// TwinCAT 3 PLC project FrameworkUnitTest
// ProgramVersion: 3.1.4026.24
// libraries:
//   [RobustSolution], * (BATW)
//   Tc2_MC2, * (Beckhoff Automation GmbH)
//   Tc2_Standard, * (Beckhoff Automation GmbH)
//   Tc2_System, * (Beckhoff Automation GmbH)
//   Tc2_Utilities, * (Beckhoff Automation GmbH)
//   Tc3_JsonXml, * (Beckhoff Automation GmbH)
//   TcUnit, * (www.tcunit.org)
// project tree:
//   DUTs/ E_FakeAxisOperation.TcDUT, ST_FakeAxisCall.TcDUT, ST_FakeAxisScriptStep.TcDUT, ST_ReferencePortTestBranch.TcDUT, ST_TestModuleFixture.TcDUT, ST_TestServiceParam.TcDUT
//   GVLs/ GVL_TestConfig.TcGVL, GVL_TestSymbols.TcGVL
//   Fakes/ FB_FakeAxis_BaseUnit.TcPOU, FB_FakeBaseUnit.TcPOU, FB_FakeHookValueReader.TcPOU, FB_FakeModuleConfigurationAdapter.TcPOU, FB_FakeModuleReferenceBindings.TcPOU, FB_FakeVariableNodeReader.TcPOU, FB_ReferencePortFixture.TcPOU, FB_TestApplicationConfigRoot.TcPOU, FB_TestableCarryoverSubStateService.TcPOU, FB_TestableHookModule.TcPOU, FB_TestableModuleBase.TcPOU, FB_TestableServiceBase.TcPOU, FB_TestCompositeService.TcPOU, FB_TestPackMLBase.TcPOU, FB_TestPackMLModeSet.TcPOU
//   POUs/Test Suites/BaseUnit/ FB_Axis_BaseUnitTests.TcPOU, FB_BaseUnitTests.TcPOU, FB_FakeAxis_BaseUnitTests.TcPOU
//   POUs/Test Suites/Configuration/ FB_ApplicationConfigRootTests.TcPOU, FB_ConfigValueSnapshotReaderTests.TcPOU, FB_LinkVariableManagerTests.TcPOU, FB_ModuleConfigurationManagerTests.TcPOU, FB_ModuleReferenceBindingContextTests.TcPOU, FB_ModuleTypeRegistryTests.TcPOU, FB_ReferenceManagerTests.TcPOU
//   POUs/Test Suites/Infrastructure/ FB_UtcClockTests.TcPOU
//   POUs/Test Suites/Module/ FB_ModuleAlarmManagerTests.TcPOU, FB_ModuleBaseTests.TcPOU
//   POUs/Test Suites/PackML/ FB_PackMLBaseTests.TcPOU, FB_PackMLModeSetTests.TcPOU
//   POUs/Test Suites/Service/ FB_CompositeServiceBaseTests.TcPOU, FB_ServiceBaseTests.TcPOU, FB_ServiceCallerTests.TcPOU, FB_ServiceCoordinatorTests.TcPOU, FB_ServiceExecuteSubStateTests.TcPOU, FB_SetMaterialServiceTests.TcPOU
//   / PlcTask.TcTTO
//   POUs/ TEST_PROG.TcPOU
// (motion and I/O tree: see PLC project robustsolutionframework)
// real-time tasks:
//   TASK UnitTest Task: cycle T#10ms, priority 21, ADS port 351
//   TASK DemoProject Task: cycle T#10ms, priority 22, ADS port 352
// variable links:

CONFIGURATION FrameworkUnitTest
    RESOURCE PLC ON TwinCAT3
        TASK PlcTask(INTERVAL := T#10ms, PRIORITY := 21);
        PROGRAM TEST_PROG WITH PlcTask : TEST_PROG;
    END_RESOURCE
END_CONFIGURATION

// ---- DUTs/E_FakeAxisOperation.TcDUT
{attribute 'qualified_only'}
{attribute 'to_string'}
TYPE E_FakeAxisOperation :
(
None := 0,
Jog,
MoveAbs,
MoveVel,
Stop,
Reset,
Halt
) UINT;
END_TYPE

// ---- DUTs/ST_FakeAxisCall.TcDUT
TYPE ST_FakeAxisCall :
STRUCT
Sequence : UDINT;
Cycle : UDINT;
Operation : E_FakeAxisOperation;
OwnerId : T_ResourceOwnerId;
Accepted : BOOL;
Execute : BOOL;
JogForward : BOOL;
JogBackwards : BOOL;
Mode : E_JogMode;
Direction : MC_Direction;
Position : LREAL;
Velocity : LREAL;
Acceleration : LREAL;
Deceleration : LREAL;
END_STRUCT
END_TYPE

// ---- DUTs/ST_FakeAxisScriptStep.TcDUT
TYPE ST_FakeAxisScriptStep :
STRUCT
Operation : E_FakeAxisOperation;
AfterActiveCycles : UINT;
Done : BOOL;
InVelocity : BOOL;
Error : BOOL;
ErrorId : UDINT;
Started : BOOL;
ResultLatched : BOOL;
Consumed : BOOL;
ActiveCycles : UINT;
END_STRUCT
END_TYPE

// ---- DUTs/ST_ReferencePortTestBranch.TcDUT
TYPE ST_ReferencePortTestBranch :
STRUCT
Axis : I_Axis_BaseUnit;
Axes : ARRAY[1..2] OF I_Axis_BaseUnit;
PortWithAnIntentionallyLongNameForReferenceBindingTests : I_Axis_BaseUnit;
END_STRUCT
END_TYPE

// ---- DUTs/ST_TestModuleFixture.TcDUT
TYPE ST_TestModuleFixture :
STRUCT
InputBool : BOOL;
OutputBool : BOOL;
SignedValue : DINT;
UnsignedValue : UDINT;
RealValue : REAL;
LongRealValue : LREAL;
TextValue : STRING(80);
BaseUnitPort : I_BaseUnit;
Nested : ST_ReferencePortTestBranch;
END_STRUCT
END_TYPE

// ---- DUTs/ST_TestServiceParam.TcDUT
TYPE ST_TestServiceParam :
STRUCT
// 使用兩個欄位，確保 Tc3_JsonXml 能反查真實 DUT 型別名稱。
Value : DINT;
Sequence : UDINT;
END_STRUCT
END_TYPE

// ---- GVLs/GVL_TestConfig.TcGVL
{attribute 'qualified_only'}
VAR_GLOBAL CONSTANT
// 預設不註冊需要外部 NC 與測試檔案的案例，避免把缺少前置條件誤報為成功。
RunNcAxisRuntimeTests : BOOL := FALSE;
RunConfigurationFileRuntimeTests : BOOL := TRUE;
ConfigurationFixtureRoot : STRING(255) := 'C:\ProgramData\RobustSolution\Tests\';
END_VAR

// ---- GVLs/GVL_TestSymbols.TcGVL
{attribute 'qualified_only'}
VAR_GLOBAL
// 具名全域變數會產生 ADS symbol，供 symbol/reflection 相關 runtime 測試使用。
InfrastructureBool : BOOL;
InfrastructureOutputBool : BOOL;
InfrastructureDInt : DINT;
InfrastructureLReal : LREAL;
InfrastructureText : STRING(80);
ModuleOne : ST_TestModuleFixture;
ModuleTwo : ST_TestModuleFixture;
RegisteredBaseUnit : FB_BaseUnit;
SecondaryBaseUnit : FB_BaseUnit;
UnprovidedBaseUnit : FB_FakeBaseUnit;
END_VAR

// ---- POUs/TEST_PROG.TcPOU
PROGRAM TEST_PROG
VAR
	BaseUnitTests : FB_BaseUnitTests;
	AxisBaseUnitTests : FB_Axis_BaseUnitTests;
	FakeAxisContractTests : FB_FakeAxis_BaseUnitTests;
	UtcClockTests : FB_UtcClockTests;
	PackMLBaseTests : FB_PackMLBaseTests;
	PackMLModeSetTests : FB_PackMLModeSetTests;
	ServiceBaseTests : FB_ServiceBaseTests;
	ServiceExecuteSubStateTests : FB_ServiceExecuteSubStateTests;
	CompositeServiceBaseTests : FB_CompositeServiceBaseTests;
	SetMaterialServiceTests : FB_SetMaterialServiceTests;
	ServiceCallerTests : FB_ServiceCallerTests;
	ServiceCoordinatorTests : FB_ServiceCoordinatorTests;
	ModuleAlarmManagerTests : FB_ModuleAlarmManagerTests;
	ModuleBaseTests : FB_ModuleBaseTests;
	ConfigValueSnapshotReaderTests : FB_ConfigValueSnapshotReaderTests;
	LinkVariableManagerTests : FB_LinkVariableManagerTests;
	ReferenceManagerTests : FB_ReferenceManagerTests;
	ModuleReferenceBindingContextTests : FB_ModuleReferenceBindingContextTests;
	ModuleTypeRegistryTests : FB_ModuleTypeRegistryTests;
	ModuleConfigurationManagerTests : FB_ModuleConfigurationManagerTests;
	ApplicationConfigRootTests : FB_ApplicationConfigRootTests;
END_VAR

// 上述 FB_TestSuite instances 會向 TcUnit 註冊；runner 每個週期統一驅動測試。
TcUnit.RUN();

END_PROGRAM

// ---- POUs/Test Suites/BaseUnit/FB_BaseUnitTests.TcPOU
FUNCTION_BLOCK FB_BaseUnitTests EXTENDS TcUnit.FB_TestSuite
VAR
	_BaseUnit : FB_BaseUnit;
END_VAR

InitialStateAndZeroOwnerAreSafe();
OwnershipIsExclusiveAndReleaseIsOwnerOnly();
AdsMetadataDescribesTheInstance();

METHOD InitialStateAndZeroOwnerAreSafe
TEST('InitialStateAndZeroOwnerAreSafe');

// Arrange：新建立的 BaseUnit 尚未被任何 Service 占用。
// Act / Assert：OwnerId=0 代表未占用，永遠不能取得、擁有或釋放資源。
AssertFalse(
	Condition := _BaseUnit.ResourceIsAcquired,
	Message := 'A new BaseUnit must be unowned.'
);
AssertTrue(
	Condition := _BaseUnit.ResourceOwnerId = 0,
	Message := 'The unowned sentinel must be zero.'
);
AssertFalse(
	Condition := _BaseUnit.M_AcquireResource(OwnerId := 0),
	Message := 'Owner zero must not acquire a resource.'
);
AssertFalse(
	Condition := _BaseUnit.M_IsResourceOwner(OwnerId := 0),
	Message := 'Owner zero must never be reported as owner.'
);
AssertFalse(
	Condition := _BaseUnit.M_ReleaseResource(OwnerId := 0),
	Message := 'Owner zero must not release a resource.'
);

TEST_FINISHED();
END_METHOD

METHOD OwnershipIsExclusiveAndReleaseIsOwnerOnly
TEST('OwnershipIsExclusiveAndReleaseIsOwnerOnly');

// Arrange / Act：Owner 11 先取得資源；同 Owner 重入應維持冪等。
AssertTrue(
	Condition := _BaseUnit.M_AcquireResource(OwnerId := 11),
	Message := 'The first valid owner must acquire the resource.'
);
AssertTrue(
	Condition := _BaseUnit.M_AcquireResource(OwnerId := 11),
	Message := 'Re-acquiring by the owner must be idempotent.'
);

// Assert：競爭者不能取得或釋放；目前 Owner 可正常釋放。
AssertFalse(
	Condition := _BaseUnit.M_AcquireResource(OwnerId := 12),
	Message := 'A competing owner must be rejected.'
);
AssertFalse(
	Condition := _BaseUnit.M_ReleaseResource(OwnerId := 12),
	Message := 'A non-owner must not release the resource.'
);
AssertTrue(
	Condition := _BaseUnit.ResourceIsAcquired AND (_BaseUnit.ResourceOwnerId = 11),
	Message := 'Rejected operations must preserve ownership.'
);
AssertTrue(
	Condition := _BaseUnit.M_ReleaseResource(OwnerId := 11),
	Message := 'The current owner must release the resource.'
);
AssertFalse(
	Condition := _BaseUnit.ResourceIsAcquired,
	Message := 'Release must restore the unowned state.'
);

TEST_FINISHED();
END_METHOD

METHOD AdsMetadataDescribesTheInstance
VAR
	pData : PVOID;
	nData : UDINT;
END_VAR
TEST('AdsMetadataDescribesTheInstance');

// Act：取得 framework 對外提供的 ADS metadata。
AssertTrue(
	Condition := _BaseUnit.M_GetAdsSymbolMetadata(Address => pData, Size => nData),
	Message := 'BaseUnit metadata must be available.'
);

// Assert：位址必須指向目前 instance，大小必須涵蓋整個 FB。
AssertTrue(
	Condition := pData = ADR(_BaseUnit),
	Message := 'Metadata address must identify this BaseUnit instance.'
);
AssertTrue(
	Condition := nData = SIZEOF(_BaseUnit),
	Message := 'Metadata size must match the BaseUnit instance.'
);

TEST_FINISHED();
END_METHOD

END_FUNCTION_BLOCK

// ---- POUs/Test Suites/BaseUnit/FB_Axis_BaseUnitTests.TcPOU
FUNCTION_BLOCK FB_Axis_BaseUnitTests EXTENDS TcUnit.FB_TestSuite
VAR
	_Axis : FB_Axis_BaseUnit;
END_VAR

AllMotionCommandsRejectNonOwners();
InitialAxisFeedbackIsNeutral();
NcAxisLifecycleRequiresExplicitRuntimeOptIn();

METHOD AllMotionCommandsRejectNonOwners
VAR
	bDone : BOOL;
	bInVelocity : BOOL;
	bError : BOOL;
	nErrorId : UDINT;
END_VAR
TEST('AllMotionCommandsRejectNonOwners');

// Arrange：不先取得 ownership，避免任何 MC function block 被啟動。
// Act / Assert：六種命令都必須在 ownership gate 被拒絕，輸出保持中性。
AssertFalse(
	Condition := _Axis.M_Halt(
		OwnerId := 1,
		Execute := TRUE,
		Deceleration := 1,
		Done => bDone,
		Error => bError
	),
	Message := 'Halt must reject a non-owner.'
);
AssertFalse(
	Condition := bDone OR bError,
	Message := 'Rejected Halt outputs must be neutral.'
);
AssertFalse(
	Condition := _Axis.M_Jog(
		OwnerId := 1,
		JogForward := TRUE,
		JogBackwards := FALSE,
		Mode := E_JogMode.MC_JOGMODE_CONTINOUS,
		Position := 0,
		Velocity := 1,
		Acceleration := 1,
		Deceleration := 1,
		Done => bDone,
		Error => bError,
		ErrorId => nErrorId
	),
	Message := 'Jog must reject a non-owner.'
);
AssertFalse(
	Condition := bDone OR bError OR (nErrorId <> 0),
	Message := 'Rejected Jog outputs must be neutral.'
);
AssertFalse(
	Condition := _Axis.M_MoveAbs(
		OwnerId := 1,
		Execute := TRUE,
		Position := 1,
		Velocity := 1,
		Acceleration := 1,
		Deceleration := 1,
		Done => bDone,
		Error => bError,
		ErrorId => nErrorId
	),
	Message := 'MoveAbs must reject a non-owner.'
);
AssertFalse(
	Condition := _Axis.M_MoveVel(
		OwnerId := 1,
		Execute := TRUE,
		Direction := MC_Direction.MC_Positive_Direction,
		Velocity := 1,
		Acceleration := 1,
		Deceleration := 1,
		InVelocity => bInVelocity,
		Error => bError
	),
	Message := 'MoveVel must reject a non-owner.'
);
AssertFalse(
	Condition := _Axis.M_Reset(
		OwnerId := 1,
		Execute := TRUE,
		Done => bDone,
		Error => bError,
		ErrorId => nErrorId
	),
	Message := 'Reset must reject a non-owner.'
);
AssertFalse(
	Condition := _Axis.M_Stop(
		OwnerId := 1,
		Execute := TRUE,
		Deceleration := 1,
		Done => bDone,
		Error => bError,
		ErrorId => nErrorId
	),
	Message := 'Stop must reject a non-owner.'
);

TEST_FINISHED();
END_METHOD

METHOD InitialAxisFeedbackIsNeutral
TEST('InitialAxisFeedbackIsNeutral');

// Assert：未連結 NC 軸時，只驗證不需驅動硬體的公開 feedback 初值。
AssertTrue(
	Condition := (_Axis.AxisActualPosition = 0.0) AND (_Axis.AxisActualVelocity = 0.0),
	Message := 'Unlinked Axis feedback must start at zero.'
);
AssertFalse(
	Condition := _Axis.AxisHasJob,
	Message := 'An unlinked Axis must not report a job.'
);

TEST_FINISHED();
END_METHOD

METHOD NcAxisLifecycleRequiresExplicitRuntimeOptIn
VAR
	bDone : BOOL;
	bError : BOOL;
	nErrorId : UDINT;
END_VAR
// RuntimeDependent：未在 XAE 將此 instance 的 _Axis 連到模擬 NC 軸時，不註冊這個 TcUnit case。
IF NOT GVL_TestConfig.RunNcAxisRuntimeTests THEN
	RETURN;
END_IF
TEST('NcAxisLifecycleRequiresExplicitRuntimeOptIn');

// Arrange：XAE 中已完成模擬 NC 軸連結，且測試開關明確設為 TRUE。
AssertTrue(
	Condition := _Axis.M_AcquireResource(OwnerId := 77),
	Message := 'Runtime owner must acquire the Axis.'
);

// Act：Reset 命令由真實 MC_Reset 執行；多掃描完成狀態由目標 Runtime 驗證。
AssertTrue(
	Condition := _Axis.M_Reset(
		OwnerId := 77,
		Execute := TRUE,
		Done => bDone,
		Error => bError,
		ErrorId => nErrorId
	),
	Message := 'Owned Reset must reach the MC layer.'
);
_Axis.M_CyclicUpdate();
AssertFalse(
	Condition := bDone AND bError,
	Message := 'MC Reset must never report Done and Error together.'
);

TEST_FINISHED();
END_METHOD

END_FUNCTION_BLOCK

// ---- POUs/Test Suites/BaseUnit/FB_FakeAxis_BaseUnitTests.TcPOU
FUNCTION_BLOCK FB_FakeAxis_BaseUnitTests EXTENDS TcUnit.FB_TestSuite
VAR
	_FakeAxis : FB_FakeAxis_BaseUnit;
	_Axis : I_Axis_BaseUnit;
END_VAR

ResourceCanBeAcquiredAndReleased();
OwnerZeroAndNonOwnerStopAreRejected();
AllNonOwnerMotionCommandsAreRejected();
ValidOwnerHaltIsAcceptedAndRecorded();
OwnerZeroAndNonOwnerHaltAreRejected();
HaltDoneIsPublishedAfterConfiguredCycles();
HaltErrorIsPublishedAfterConfiguredCycles();
HaltWithdrawalClearsResultAndPreservesOwnership();
ScriptAndHistoryOverflowAreExplicit();
CommandHistoryPreservesParameters();
ResponseRemainsLatchedUntilCommandWithdrawal();
JogErrorIsPublishedAfterConfiguredCycles();
ActualFeedbackIsAvailableThroughInterface();

METHOD ActualFeedbackIsAvailableThroughInterface
VAR
	FakeAxis : FB_FakeAxis_BaseUnit;
	Axis : I_Axis_BaseUnit;
END_VAR
TEST('ActualFeedbackIsAvailableThroughInterface');

FakeAxis.M_ResetScenario();
FakeAxis.M_SetAxisFeedback(ActualPosition := 45.25, ActualVelocity := 123.5);
Axis := FakeAxis;

AssertTrue(
	Condition := Axis.AxisActualPosition = 45.25,
	Message := 'Axis interface must expose actual position feedback.'
);
AssertTrue(
	Condition := Axis.AxisActualVelocity = 123.5,
	Message := 'Axis interface must expose actual velocity feedback.'
);

TEST_FINISHED();
END_METHOD

METHOD AllNonOwnerMotionCommandsAreRejected
VAR
	bDone : BOOL;
	bInVelocity : BOOL;
	bError : BOOL;
	nErrorId : UDINT;
END_VAR
TEST('AllNonOwnerMotionCommandsAreRejected');

_FakeAxis.M_ResetScenario();
_Axis := _FakeAxis;
AssertTrue(
	Condition := _Axis.M_AcquireResource(OwnerId := 1),
	Message := 'Owner 1 must acquire the Axis.'
);
AssertFalse(
	Condition := _Axis.M_Jog(
		OwnerId := 2,
		JogForward := TRUE,
		JogBackwards := FALSE,
		Mode := E_JogMode.MC_JOGMODE_CONTINOUS,
		Position := 1,
		Velocity := 2,
		Acceleration := 3,
		Deceleration := 4,
		Done => bDone,
		Error => bError,
		ErrorId => nErrorId
	),
	Message := 'Non-Owner Jog must be rejected.'
);
AssertFalse(
	Condition := bDone OR bError OR (nErrorId <> 0),
	Message := 'Rejected Jog outputs must be neutral.'
);
AssertFalse(
	Condition := _Axis.M_MoveAbs(
		OwnerId := 2,
		Execute := TRUE,
		Position := 1,
		Velocity := 2,
		Acceleration := 3,
		Deceleration := 4,
		Done => bDone,
		Error => bError
	),
	Message := 'Non-Owner MoveAbs must be rejected.'
);
AssertFalse(
	Condition := _Axis.M_MoveVel(
		OwnerId := 2,
		Execute := TRUE,
		Direction := MC_Direction.MC_Positive_Direction,
		Velocity := 2,
		Acceleration := 3,
		Deceleration := 4,
		InVelocity => bInVelocity,
		Error => bError
	),
	Message := 'Non-Owner MoveVel must be rejected.'
);
AssertFalse(
	Condition := _Axis.M_Reset(
		OwnerId := 2,
		Execute := TRUE,
		Done => bDone,
		Error => bError
	),
	Message := 'Non-Owner Reset must be rejected.'
);
AssertFalse(
	Condition := bDone OR bInVelocity OR bError,
	Message := 'All rejected motion outputs must remain neutral.'
);

TEST_FINISHED();
END_METHOD

METHOD CommandHistoryPreservesParameters
VAR
	CallRecord : ST_FakeAxisCall;
END_VAR
TEST('CommandHistoryPreservesParameters');

_FakeAxis.M_ResetScenario();
_Axis := _FakeAxis;
AssertTrue(
	Condition := _Axis.M_AcquireResource(OwnerId := 5),
	Message := 'History test Owner must acquire Axis.'
);
_Axis.M_MoveAbs(
	OwnerId := 5,
	Execute := TRUE,
	Position := 123.5,
	Velocity := 45.5,
	Acceleration := 67.5,
	Deceleration := 89.5
);
AssertTrue(
	Condition := _FakeAxis.M_GetCall(Index := 1, CallRecord => CallRecord),
	Message := 'Accepted MoveAbs must be present in history.'
);
AssertTrue(
	Condition := CallRecord.Accepted AND CallRecord.Execute,
	Message := 'History must retain acceptance and Execute.'
);
AssertTrue(
	Condition :=
		(CallRecord.Position = 123.5)
		AND (CallRecord.Velocity = 45.5)
		AND (CallRecord.Acceleration = 67.5)
		AND (CallRecord.Deceleration = 89.5),
	Message := 'History must retain all motion parameters.'
);

_Axis.M_MoveAbs(
	OwnerId := 6,
	Execute := FALSE,
	Position := 1,
	Velocity := 2,
	Acceleration := 3,
	Deceleration := 4
);
AssertTrue(
	Condition := _FakeAxis.M_GetCall(Index := 2, CallRecord => CallRecord),
	Message := 'Rejected command must still be recorded.'
);
AssertFalse(
	Condition := CallRecord.Accepted,
	Message := 'Rejected history entry must be marked rejected.'
);
AssertTrue(
	Condition := CallRecord.Sequence = 2,
	Message := 'History sequence must be global and monotonic.'
);

TEST_FINISHED();
END_METHOD

METHOD HaltDoneIsPublishedAfterConfiguredCycles
VAR_INST
	FakeAxis : FB_FakeAxis_BaseUnit;
	Axis : I_Axis_BaseUnit;
	nPhase : UINT;
	bDone : BOOL;
	bError : BOOL;
END_VAR
TEST('HaltDoneIsPublishedAfterConfiguredCycles');

CASE nPhase OF
	0:
		FakeAxis.M_ResetScenario();
		Axis := FakeAxis;
		AssertTrue(
			Condition := Axis.M_AcquireResource(OwnerId := 21),
			Message := 'Halt Done test Owner must acquire the Axis.'
		);
		AssertTrue(
			Condition := FakeAxis.M_QueueResult(
				Operation := E_FakeAxisOperation.Halt,
				AfterActiveCycles := 2,
				Done := TRUE,
				InVelocity := FALSE,
				Error := FALSE,
				ErrorId := 0
			),
			Message := 'Halt Done script must be queued.'
		);
		AssertTrue(
			Condition := Axis.M_Halt(
				OwnerId := 21,
				Execute := TRUE,
				Deceleration := 10,
				Done => bDone,
				Error => bError
			),
			Message := 'Owner Halt must be accepted.'
		);
		AssertFalse(
			Condition := bDone OR bError,
			Message := 'Halt result must initially be pending.'
		);
		nPhase := 1;

	1:
		Axis.M_CyclicUpdate();
		Axis.M_Halt(
			OwnerId := 21,
			Execute := TRUE,
			Deceleration := 10,
			Done => bDone,
			Error => bError
		);
		AssertFalse(
			Condition := bDone OR bError,
			Message := 'Halt Done must remain pending after one active cycle.'
		);
		nPhase := 2;

	2:
		Axis.M_CyclicUpdate();
		Axis.M_Halt(
			OwnerId := 21,
			Execute := TRUE,
			Deceleration := 10,
			Done => bDone,
			Error => bError
		);
		AssertTrue(
			Condition := bDone AND NOT bError,
			Message := 'Halt Done must be published on the configured cycle.'
		);
		nPhase := 0;
		TEST_FINISHED();
END_CASE
END_METHOD

METHOD HaltErrorIsPublishedAfterConfiguredCycles
VAR_INST
	FakeAxis : FB_FakeAxis_BaseUnit;
	Axis : I_Axis_BaseUnit;
	nPhase : UINT;
	bDone : BOOL;
	bError : BOOL;
END_VAR
TEST('HaltErrorIsPublishedAfterConfiguredCycles');

CASE nPhase OF
	0:
		FakeAxis.M_ResetScenario();
		Axis := FakeAxis;
		AssertTrue(
			Condition := Axis.M_AcquireResource(OwnerId := 22),
			Message := 'Halt Error test Owner must acquire the Axis.'
		);
		AssertTrue(
			Condition := FakeAxis.M_QueueResult(
				Operation := E_FakeAxisOperation.Halt,
				AfterActiveCycles := 2,
				Done := FALSE,
				InVelocity := FALSE,
				Error := TRUE,
				ErrorId := 16#5678
			),
			Message := 'Halt Error script must be queued.'
		);
		Axis.M_Halt(
			OwnerId := 22,
			Execute := TRUE,
			Deceleration := 11,
			Done => bDone,
			Error => bError
		);
		AssertFalse(
			Condition := bDone OR bError,
			Message := 'Halt Error must initially be pending.'
		);
		nPhase := 1;

	1:
		Axis.M_CyclicUpdate();
		Axis.M_Halt(
			OwnerId := 22,
			Execute := TRUE,
			Deceleration := 11,
			Done => bDone,
			Error => bError
		);
		AssertFalse(
			Condition := bDone OR bError,
			Message := 'Halt Error must remain pending after one active cycle.'
		);
		nPhase := 2;

	2:
		Axis.M_CyclicUpdate();
		Axis.M_Halt(
			OwnerId := 22,
			Execute := TRUE,
			Deceleration := 11,
			Done => bDone,
			Error => bError
		);
		AssertTrue(
			Condition := bError AND NOT bDone,
			Message := 'Halt Error must be published on the configured cycle.'
		);
		nPhase := 0;
		TEST_FINISHED();
END_CASE
END_METHOD

METHOD HaltWithdrawalClearsResultAndPreservesOwnership
VAR_INST
	FakeAxis : FB_FakeAxis_BaseUnit;
	Axis : I_Axis_BaseUnit;
	nPhase : UINT;
	bDone : BOOL;
	bError : BOOL;
	CallRecord : ST_FakeAxisCall;
END_VAR
TEST('HaltWithdrawalClearsResultAndPreservesOwnership');

CASE nPhase OF
	0:
		FakeAxis.M_ResetScenario();
		Axis := FakeAxis;
		AssertTrue(
			Condition := Axis.M_AcquireResource(OwnerId := 23),
			Message := 'Halt withdrawal test Owner must acquire the Axis.'
		);
		AssertTrue(
			Condition := FakeAxis.M_QueueResult(
				Operation := E_FakeAxisOperation.Halt,
				AfterActiveCycles := 1,
				Done := TRUE,
				InVelocity := FALSE,
				Error := FALSE,
				ErrorId := 0
			),
			Message := 'Halt withdrawal script must be queued.'
		);
		Axis.M_Halt(OwnerId := 23, Execute := TRUE, Deceleration := 12);
		nPhase := 1;

	1:
		Axis.M_CyclicUpdate();
		Axis.M_Halt(
			OwnerId := 23,
			Execute := TRUE,
			Deceleration := 12,
			Done => bDone,
			Error => bError
		);
		AssertTrue(
			Condition := bDone AND NOT bError,
			Message := 'Halt must complete before command withdrawal.'
		);
		AssertTrue(
			Condition := Axis.M_IsResourceOwner(OwnerId := 23),
			Message := 'Halt completion must not release its Owner.'
		);
		AssertTrue(
			Condition := Axis.M_Halt(OwnerId := 23, Execute := FALSE, Deceleration := 12),
			Message := 'Owner must be allowed to withdraw Halt.'
		);
		AssertTrue(
			Condition := FakeAxis.M_GetCall(Index := 3, CallRecord => CallRecord),
			Message := 'Withdrawn Halt must be recorded.'
		);
		AssertTrue(
			Condition :=
				(CallRecord.Operation = E_FakeAxisOperation.Halt)
				AND CallRecord.Accepted
				AND NOT CallRecord.Execute,
			Message := 'Halt history must expose accepted command withdrawal.'
		);
		Axis.M_CyclicUpdate();
		nPhase := 2;

	2:
		Axis.M_Halt(
			OwnerId := 23,
			Execute := FALSE,
			Deceleration := 12,
			Done => bDone,
			Error => bError
		);
		AssertFalse(
			Condition := bDone OR bError,
			Message := 'Halt result must clear after withdrawal and cyclic update.'
		);
		AssertTrue(
			Condition := Axis.M_IsResourceOwner(OwnerId := 23),
			Message := 'Halt withdrawal must preserve resource ownership.'
		);
		AssertFalse(
			Condition := Axis.M_AcquireResource(OwnerId := 24),
			Message := 'A contender must remain rejected after Halt withdrawal.'
		);
		nPhase := 0;
		TEST_FINISHED();
END_CASE
END_METHOD

METHOD JogErrorIsPublishedAfterConfiguredCycles
VAR_INST
	FakeAxis : FB_FakeAxis_BaseUnit;
	Axis : I_Axis_BaseUnit;
	nPhase : UINT;
	bError : BOOL;
	bQueued : BOOL;
END_VAR
TEST('JogErrorIsPublishedAfterConfiguredCycles');

CASE nPhase OF
	0:
		FakeAxis.M_ResetScenario();
		Axis := FakeAxis;
		AssertTrue(
			Condition := Axis.M_AcquireResource(OwnerId := 1),
			Message := 'Test Owner must acquire the Axis.'
		);
		bQueued := FakeAxis.M_QueueResult(
			Operation := E_FakeAxisOperation.Jog,
			AfterActiveCycles := 2,
			Done := FALSE,
			InVelocity := FALSE,
			Error := TRUE,
			ErrorId := 16#1234);
		AssertTrue(Condition := bQueued, Message := 'A valid Jog Error script must be queued.');
		Axis.M_Jog(
			OwnerId := 1,
			JogForward := TRUE,
			JogBackwards := FALSE,
			Mode := E_JogMode.MC_JOGMODE_CONTINOUS,
			Position := 0,
			Velocity := 10,
			Acceleration := 20,
			Deceleration := 30);
		nPhase := 1;

	1:
		Axis.M_CyclicUpdate();
		Axis.M_Jog(
			OwnerId := 1,
			JogForward := TRUE,
			JogBackwards := FALSE,
			Mode := E_JogMode.MC_JOGMODE_CONTINOUS,
			Position := 0,
			Velocity := 10,
			Acceleration := 20,
			Deceleration := 30,
			Error => bError);
		AssertFalse(
			Condition := bError,
			Message := 'Jog Error must remain pending after one active cycle.'
		);
		nPhase := 2;

	2:
		Axis.M_CyclicUpdate();
		Axis.M_Jog(
			OwnerId := 1,
			JogForward := TRUE,
			JogBackwards := FALSE,
			Mode := E_JogMode.MC_JOGMODE_CONTINOUS,
			Position := 0,
			Velocity := 10,
			Acceleration := 20,
			Deceleration := 30,
			Error => bError);
		AssertTrue(
			Condition := bError,
			Message := 'Jog Error must be published on the configured cycle.'
		);
		nPhase := 0;
		TEST_FINISHED();
END_CASE
END_METHOD

METHOD OwnerZeroAndNonOwnerHaltAreRejected
VAR
	bDone : BOOL;
	bError : BOOL;
	bAccepted : BOOL;
	CallRecord : ST_FakeAxisCall;
END_VAR
TEST('OwnerZeroAndNonOwnerHaltAreRejected');

_FakeAxis.M_ResetScenario();
_Axis := _FakeAxis;
AssertTrue(
	Condition := _Axis.M_AcquireResource(OwnerId := 31),
	Message := 'Valid Owner must acquire the Axis.'
);

bAccepted := _Axis.M_Halt(
	OwnerId := 0,
	Execute := TRUE,
	Deceleration := 20,
	Done => bDone,
	Error => bError
);
AssertFalse(Condition := bAccepted, Message := 'OwnerId zero Halt must be rejected.');
AssertFalse(
	Condition := bDone OR bError,
	Message := 'OwnerId zero Halt outputs must be neutral.'
);
AssertTrue(
	Condition := _FakeAxis.M_GetCall(Index := 1, CallRecord => CallRecord),
	Message := 'OwnerId zero Halt must be recorded.'
);
AssertFalse(
	Condition := CallRecord.Accepted,
	Message := 'OwnerId zero Halt history must be rejected.'
);

bAccepted := _Axis.M_Halt(
	OwnerId := 32,
	Execute := TRUE,
	Deceleration := 21,
	Done => bDone,
	Error => bError
);
AssertFalse(Condition := bAccepted, Message := 'Non-Owner Halt must be rejected.');
AssertFalse(
	Condition := bDone OR bError,
	Message := 'Non-Owner Halt outputs must be neutral.'
);
AssertTrue(
	Condition := _FakeAxis.M_GetCall(Index := 2, CallRecord => CallRecord),
	Message := 'Non-Owner Halt must be recorded.'
);
AssertFalse(
	Condition := CallRecord.Accepted,
	Message := 'Non-Owner Halt history must be rejected.'
);
AssertTrue(
	Condition := _Axis.M_IsResourceOwner(OwnerId := 31),
	Message := 'Rejected Halt must preserve the current Owner.'
);

TEST_FINISHED();
END_METHOD

METHOD OwnerZeroAndNonOwnerStopAreRejected
VAR
	bDone : BOOL;
	bError : BOOL;
	bRejected : BOOL;
	bAccepted : BOOL;
END_VAR
TEST('OwnerZeroAndNonOwnerStopAreRejected');

_FakeAxis.M_ResetScenario();
_Axis := _FakeAxis;
AssertFalse(
	Condition := _Axis.M_AcquireResource(OwnerId := 0),
	Message := 'OwnerId zero must never acquire a resource.'
);
AssertTrue(
	Condition := _Axis.M_AcquireResource(OwnerId := 1),
	Message := 'Valid Owner must acquire the Axis.'
);
AssertTrue(
	Condition := _FakeAxis.M_QueueResult(
		Operation := E_FakeAxisOperation.Stop,
		AfterActiveCycles := 1,
		Done := TRUE,
		InVelocity := FALSE,
		Error := FALSE,
		ErrorId := 0
	),
	Message := 'Stop Done script must be accepted.'
);

bAccepted := _Axis.M_Stop(OwnerId := 1, Execute := TRUE, Deceleration := 10);
bRejected := _Axis.M_Stop(
	OwnerId := 2,
	Execute := FALSE,
	Deceleration := 99,
	Done => bDone,
	Error => bError
);
AssertFalse(Condition := bRejected, Message := 'Non-Owner Stop must be rejected.');
AssertFalse(
	Condition := bDone OR bError,
	Message := 'Rejected Stop must return neutral outputs.'
);

_Axis.M_CyclicUpdate();
_Axis.M_Stop(
	OwnerId := 1,
	Execute := TRUE,
	Deceleration := 10,
	Done => bDone,
	Error => bError
);
AssertTrue(
	Condition := bAccepted AND bDone AND NOT bError,
	Message := 'Rejected Stop must not cancel the active Owner command.'
);

TEST_FINISHED();
END_METHOD

METHOD ResourceCanBeAcquiredAndReleased
VAR
	bAcquired : BOOL;
	bContenderAcquired : BOOL;
	bReleased : BOOL;
END_VAR
TEST('ResourceCanBeAcquiredAndReleased');

_FakeAxis.M_ResetScenario();
_Axis := _FakeAxis;

bAcquired := _Axis.M_AcquireResource(OwnerId := 1);
bContenderAcquired := _Axis.M_AcquireResource(OwnerId := 2);
bReleased := _Axis.M_ReleaseResource(OwnerId := 1);

AssertTrue(
	Condition := bAcquired,
	Message := 'The first valid Owner must acquire the Axis.'
);
AssertFalse(
	Condition := bContenderAcquired,
	Message := 'A competing Owner must be rejected.'
);
AssertTrue(Condition := bReleased, Message := 'The active Owner must release the Axis.');
AssertFalse(
	Condition := _Axis.M_IsResourceOwner(OwnerId := 1),
	Message := 'The Axis must be unowned after Release.'
);

TEST_FINISHED();
END_METHOD

METHOD ResponseRemainsLatchedUntilCommandWithdrawal
VAR
	bError : BOOL;
END_VAR
TEST('ResponseRemainsLatchedUntilCommandWithdrawal');

_FakeAxis.M_ResetScenario();
_Axis := _FakeAxis;
AssertTrue(
	Condition := _Axis.M_AcquireResource(OwnerId := 1),
	Message := 'Latch test Owner must acquire Axis.'
);
AssertTrue(
	Condition := _FakeAxis.M_QueueResult(
		Operation := E_FakeAxisOperation.Jog,
		AfterActiveCycles := 1,
		Done := FALSE,
		InVelocity := FALSE,
		Error := TRUE,
		ErrorId := 1
	),
	Message := 'Jog Error script must be queued.'
);
_Axis.M_Jog(
	OwnerId := 1,
	JogForward := TRUE,
	JogBackwards := FALSE,
	Mode := E_JogMode.MC_JOGMODE_CONTINOUS,
	Position := 0,
	Velocity := 1,
	Acceleration := 1,
	Deceleration := 1
);
_Axis.M_CyclicUpdate();
_Axis.M_Jog(
	OwnerId := 1,
	JogForward := TRUE,
	JogBackwards := FALSE,
	Mode := E_JogMode.MC_JOGMODE_CONTINOUS,
	Position := 0,
	Velocity := 1,
	Acceleration := 1,
	Deceleration := 1,
	Error => bError
);
AssertTrue(Condition := bError, Message := 'Configured Error must latch.');
_Axis.M_CyclicUpdate();
_Axis.M_Jog(
	OwnerId := 1,
	JogForward := TRUE,
	JogBackwards := FALSE,
	Mode := E_JogMode.MC_JOGMODE_CONTINOUS,
	Position := 0,
	Velocity := 1,
	Acceleration := 1,
	Deceleration := 1,
	Error => bError
);
AssertTrue(
	Condition := bError,
	Message := 'Error must remain latched while Jog remains active.'
);
_Axis.M_Jog(
	OwnerId := 1,
	JogForward := FALSE,
	JogBackwards := FALSE,
	Mode := E_JogMode.MC_JOGMODE_CONTINOUS,
	Position := 0,
	Velocity := 1,
	Acceleration := 1,
	Deceleration := 1
);
_Axis.M_CyclicUpdate();
_Axis.M_Jog(
	OwnerId := 1,
	JogForward := FALSE,
	JogBackwards := FALSE,
	Mode := E_JogMode.MC_JOGMODE_CONTINOUS,
	Position := 0,
	Velocity := 1,
	Acceleration := 1,
	Deceleration := 1,
	Error => bError
);
AssertFalse(
	Condition := bError,
	Message :=
		'Error must clear after both Jog directions are withdrawn and cyclic update runs.'
);

TEST_FINISHED();
END_METHOD

METHOD ScriptAndHistoryOverflowAreExplicit
VAR
	nIndex : UINT;
	bQueued : BOOL;
END_VAR
TEST('ScriptAndHistoryOverflowAreExplicit');

_FakeAxis.M_ResetScenario();
_Axis := _FakeAxis;
FOR nIndex := 1 TO 32 DO
	bQueued := _FakeAxis.M_QueueResult(
		Operation := E_FakeAxisOperation.MoveAbs,
		AfterActiveCycles := nIndex,
		Done := TRUE,
		InVelocity := FALSE,
		Error := FALSE,
		ErrorId := 0
	);
END_FOR
bQueued := _FakeAxis.M_QueueResult(
	Operation := E_FakeAxisOperation.MoveAbs,
	AfterActiveCycles := 33,
	Done := TRUE,
	InVelocity := FALSE,
	Error := FALSE,
	ErrorId := 0
);
AssertFalse(Condition := bQueued, Message := 'Script queue must reject entry 33.');
AssertTrue(
	Condition := _FakeAxis.ScriptOverflowed,
	Message := 'Script overflow must be visible.'
);

_FakeAxis.M_ResetScenario();
bQueued := _FakeAxis.M_QueueResult(
	Operation := E_FakeAxisOperation.Jog,
	AfterActiveCycles := 1,
	Done := TRUE,
	InVelocity := FALSE,
	Error := TRUE,
	ErrorId := 0
);
AssertFalse(
	Condition := bQueued,
	Message := 'Done and Error cannot be configured together.'
);
AssertTrue(
	Condition := _FakeAxis.ScriptConfigurationError,
	Message := 'Invalid script configuration must be visible.'
);

FOR nIndex := 1 TO 257 DO
	_Axis.M_Reset(OwnerId := 77, Execute := TRUE);
END_FOR
AssertTrue(
	Condition := _FakeAxis.HistoryCount = 256,
	Message := 'History must stop at its fixed capacity.'
);
AssertTrue(
	Condition := _FakeAxis.HistoryOverflowed,
	Message := 'History overflow must be visible and must not overwrite calls.'
);

TEST_FINISHED();
END_METHOD

METHOD ValidOwnerHaltIsAcceptedAndRecorded
VAR
	bDone : BOOL;
	bError : BOOL;
	CallRecord : ST_FakeAxisCall;
END_VAR
TEST('ValidOwnerHaltIsAcceptedAndRecorded');

_FakeAxis.M_ResetScenario();
_Axis := _FakeAxis;
AssertTrue(
	Condition := _Axis.M_AcquireResource(OwnerId := 11),
	Message := 'Valid Halt Owner must acquire the Axis.'
);
AssertTrue(
	Condition := _Axis.M_Halt(
		OwnerId := 11,
		Execute := TRUE,
		Deceleration := 12.5,
		Done => bDone,
		Error => bError
	),
	Message := 'Valid Owner Halt must be accepted.'
);
AssertFalse(
	Condition := bDone OR bError,
	Message := 'Unscripted Halt outputs must be neutral.'
);
AssertTrue(
	Condition := _FakeAxis.M_GetCall(Index := 1, CallRecord => CallRecord),
	Message := 'Accepted Halt must be present in history.'
);
AssertTrue(
	Condition :=
		(CallRecord.Operation = E_FakeAxisOperation.Halt)
		AND CallRecord.Accepted
		AND CallRecord.Execute,
	Message := 'History must identify an accepted active Halt.'
);
AssertTrue(
	Condition := (CallRecord.OwnerId = 11) AND (CallRecord.Deceleration = 12.5),
	Message := 'Halt history must preserve Owner and deceleration.'
);

TEST_FINISHED();
END_METHOD

END_FUNCTION_BLOCK

// ---- Fakes/FB_FakeAxis_BaseUnit.TcPOU
FUNCTION_BLOCK FB_FakeAxis_BaseUnit EXTENDS FB_BaseUnit IMPLEMENTS I_Axis_BaseUnit
VAR
	_bAxisIsDisabled : BOOL;
	_bAxisHasJob : BOOL;
	_fAxisActualPosition : LREAL;
	_fAxisActualVelocity : LREAL;
	_nCycle : UDINT;
	_nCallSequence : UDINT;

	_aScripts : ARRAY[1..32] OF ST_FakeAxisScriptStep;
	_nScriptCount : UINT;
	_bScriptOverflowed : BOOL;
	_bScriptConfigurationError : BOOL;

	_aHistory : ARRAY[1..256] OF ST_FakeAxisCall;
	_nHistoryCount : UINT;
	_bHistoryOverflowed : BOOL;

	_bJogActive : BOOL;
	_bMoveAbsActive : BOOL;
	_bMoveVelActive : BOOL;
	_bStopActive : BOOL;
	_bResetActive : BOOL;
	_bHaltActive : BOOL;

	_bJogDone : BOOL;
	_bJogInVelocity : BOOL;
	_bJogError : BOOL;
	_nJogErrorId : UDINT;
	_bMoveAbsDone : BOOL;
	_bMoveAbsInVelocity : BOOL;
	_bMoveAbsError : BOOL;
	_nMoveAbsErrorId : UDINT;
	_bMoveVelDone : BOOL;
	_bMoveVelInVelocity : BOOL;
	_bMoveVelError : BOOL;
	_nMoveVelErrorId : UDINT;
	_bStopDone : BOOL;
	_bStopInVelocity : BOOL;
	_bStopError : BOOL;
	_nStopErrorId : UDINT;
	_bResetDone : BOOL;
	_bResetInVelocity : BOOL;
	_bResetError : BOOL;
	_nResetErrorId : UDINT;
	_bHaltDone : BOOL;
	_bHaltInVelocity : BOOL;
	_bHaltError : BOOL;
	_nHaltErrorId : UDINT;
END_VAR

M_CyclicUpdate();

PROPERTY AxisActualPosition : LREAL
GET
AxisActualPosition := _fAxisActualPosition;
END_GET
END_PROPERTY

PROPERTY AxisActualVelocity : LREAL
GET
AxisActualVelocity := _fAxisActualVelocity;
END_GET
END_PROPERTY

PROPERTY AxisHasJob : BOOL
GET
AxisHasJob := _bAxisHasJob;
END_GET
END_PROPERTY

PROPERTY AxisIsDisabled : BOOL
GET
AxisIsDisabled := _bAxisIsDisabled;
END_GET
END_PROPERTY

PROPERTY CurrentCycle : UDINT
GET
CurrentCycle := _nCycle;
END_GET
END_PROPERTY

PROPERTY HistoryCount : UINT
GET
HistoryCount := _nHistoryCount;
END_GET
END_PROPERTY

PROPERTY HistoryOverflowed : BOOL
GET
HistoryOverflowed := _bHistoryOverflowed;
END_GET
END_PROPERTY

METHOD M_ClearCallHistory
VAR_INPUT
END_VAR
MEMSET(ADR(_aHistory), 0, SIZEOF(_aHistory));
_nHistoryCount := 0;
_nCallSequence := 0;
_bHistoryOverflowed := FALSE;
END_METHOD

METHOD M_CyclicUpdate
VAR_INPUT
END_VAR
_nCycle := _nCycle + 1;

M_ProcessOperation(
	Operation := E_FakeAxisOperation.Jog,
	Active := _bJogActive,
	Done := _bJogDone,
	InVelocity := _bJogInVelocity,
	Error := _bJogError,
	ErrorId := _nJogErrorId
);
M_ProcessOperation(
	Operation := E_FakeAxisOperation.MoveAbs,
	Active := _bMoveAbsActive,
	Done := _bMoveAbsDone,
	InVelocity := _bMoveAbsInVelocity,
	Error := _bMoveAbsError,
	ErrorId := _nMoveAbsErrorId
);
M_ProcessOperation(
	Operation := E_FakeAxisOperation.MoveVel,
	Active := _bMoveVelActive,
	Done := _bMoveVelDone,
	InVelocity := _bMoveVelInVelocity,
	Error := _bMoveVelError,
	ErrorId := _nMoveVelErrorId
);
M_ProcessOperation(
	Operation := E_FakeAxisOperation.Stop,
	Active := _bStopActive,
	Done := _bStopDone,
	InVelocity := _bStopInVelocity,
	Error := _bStopError,
	ErrorId := _nStopErrorId
);
M_ProcessOperation(
	Operation := E_FakeAxisOperation.Reset,
	Active := _bResetActive,
	Done := _bResetDone,
	InVelocity := _bResetInVelocity,
	Error := _bResetError,
	ErrorId := _nResetErrorId
);
M_ProcessOperation(
	Operation := E_FakeAxisOperation.Halt,
	Active := _bHaltActive,
	Done := _bHaltDone,
	InVelocity := _bHaltInVelocity,
	Error := _bHaltError,
	ErrorId := _nHaltErrorId
);
END_METHOD

METHOD M_GetCall : BOOL
VAR_INPUT
	Index : UINT;
END_VAR
VAR_OUTPUT
	CallRecord : ST_FakeAxisCall;
END_VAR
M_GetCall := FALSE;
MEMSET(ADR(CallRecord), 0, SIZEOF(CallRecord));
IF (Index = 0) OR (Index > _nHistoryCount) THEN
	RETURN;
END_IF
CallRecord := _aHistory[Index];
M_GetCall := TRUE;
END_METHOD

METHOD M_Halt : BOOL
VAR_INPUT
	OwnerId : T_ResourceOwnerId;
	Execute : BOOL;
	Deceleration : LREAL;
END_VAR
VAR_OUTPUT
	Done : BOOL;
	Error : BOOL;
END_VAR
VAR
	bAccepted : BOOL;
END_VAR
bAccepted := M_IsResourceOwner(OwnerId := OwnerId);
M_RecordCall(
	Operation := E_FakeAxisOperation.Halt,
	OwnerId := OwnerId,
	Accepted := bAccepted,
	Execute := Execute,
	JogForward := FALSE,
	JogBackwards := FALSE,
	Mode := E_JogMode.MC_JOGMODE_CONTINOUS,
	Direction := MC_Direction.MC_Positive_Direction,
	Position := 0,
	Velocity := 0,
	Acceleration := 0,
	Deceleration := Deceleration
);

M_Halt := bAccepted;
IF NOT bAccepted THEN
	Done := FALSE;
	Error := FALSE;
	RETURN;
END_IF

_bHaltActive := Execute;
Done := _bHaltDone;
Error := _bHaltError;
END_METHOD

METHOD M_Jog : BOOL
VAR_INPUT
	OwnerId : T_ResourceOwnerId;
	JogForward : BOOL;
	JogBackwards : BOOL;
	Mode : E_JogMode;
	Position : LREAL;
	Velocity : LREAL;
	Acceleration : LREAL;
	Deceleration : LREAL;
END_VAR
VAR_OUTPUT
	Done : BOOL;
	Error : BOOL;
	ErrorId : UDINT;
END_VAR
VAR
	bAccepted : BOOL;
END_VAR
bAccepted := M_IsResourceOwner(OwnerId := OwnerId);
M_RecordCall(
	Operation := E_FakeAxisOperation.Jog,
	OwnerId := OwnerId,
	Accepted := bAccepted,
	Execute := JogForward OR JogBackwards,
	JogForward := JogForward,
	JogBackwards := JogBackwards,
	Mode := Mode,
	Direction := MC_Direction.MC_Positive_Direction,
	Position := Position,
	Velocity := Velocity,
	Acceleration := Acceleration,
	Deceleration := Deceleration
);

M_Jog := bAccepted;
IF NOT bAccepted THEN
	Done := FALSE;
	Error := FALSE;
	ErrorId := 0;
	RETURN;
END_IF

_bJogActive := JogForward OR JogBackwards;
Done := _bJogDone;
Error := _bJogError;
ErrorId := _nJogErrorId;
END_METHOD

METHOD M_MoveAbs : BOOL
VAR_INPUT
	OwnerId : T_ResourceOwnerId;
	Execute : BOOL;
	Position : LREAL;
	Velocity : LREAL;
	Acceleration : LREAL;
	Deceleration : LREAL;
END_VAR
VAR_OUTPUT
	Done : BOOL;
	Error : BOOL;
	ErrorId : UDINT;
END_VAR
VAR
	bAccepted : BOOL;
END_VAR
bAccepted := M_IsResourceOwner(OwnerId := OwnerId);
M_RecordCall(
	Operation := E_FakeAxisOperation.MoveAbs,
	OwnerId := OwnerId,
	Accepted := bAccepted,
	Execute := Execute,
	JogForward := FALSE,
	JogBackwards := FALSE,
	Mode := E_JogMode.MC_JOGMODE_CONTINOUS,
	Direction := MC_Direction.MC_Positive_Direction,
	Position := Position,
	Velocity := Velocity,
	Acceleration := Acceleration,
	Deceleration := Deceleration
);

M_MoveAbs := bAccepted;
IF NOT bAccepted THEN
	Done := FALSE;
	Error := FALSE;
	ErrorId := 0;
	RETURN;
END_IF

_bMoveAbsActive := Execute;
Done := _bMoveAbsDone;
Error := _bMoveAbsError;
ErrorId := _nMoveAbsErrorId;
END_METHOD

METHOD M_MoveVel : BOOL
VAR_INPUT
	OwnerId : T_ResourceOwnerId;
	Execute : BOOL;
	Direction : MC_Direction;
	Velocity : LREAL;
	Acceleration : LREAL;
	Deceleration : LREAL;
END_VAR
VAR_OUTPUT
	InVelocity : BOOL;
	Error : BOOL;
END_VAR
VAR
	bAccepted : BOOL;
END_VAR
bAccepted := M_IsResourceOwner(OwnerId := OwnerId);
M_RecordCall(
	Operation := E_FakeAxisOperation.MoveVel,
	OwnerId := OwnerId,
	Accepted := bAccepted,
	Execute := Execute,
	JogForward := FALSE,
	JogBackwards := FALSE,
	Mode := E_JogMode.MC_JOGMODE_CONTINOUS,
	Direction := Direction,
	Position := 0,
	Velocity := Velocity,
	Acceleration := Acceleration,
	Deceleration := Deceleration
);

M_MoveVel := bAccepted;
IF NOT bAccepted THEN
	InVelocity := FALSE;
	Error := FALSE;
	RETURN;
END_IF

_bMoveVelActive := Execute;
InVelocity := _bMoveVelInVelocity;
Error := _bMoveVelError;
END_METHOD

METHOD PRIVATE M_ProcessOperation
VAR_INPUT
	Operation : E_FakeAxisOperation;
	Active : BOOL;
END_VAR
VAR_IN_OUT
	Done : BOOL;
	InVelocity : BOOL;
	Error : BOOL;
	ErrorId : UDINT;
END_VAR
VAR
	nIndex : UINT;
END_VAR
Done := FALSE;
InVelocity := FALSE;
Error := FALSE;
ErrorId := 0;

FOR nIndex := 1 TO _nScriptCount DO
	IF (_aScripts[nIndex].Operation = Operation) AND NOT _aScripts[nIndex].Consumed THEN

		// Label script that is consumed
		IF NOT Active THEN
			IF _aScripts[nIndex].Started THEN
				_aScripts[nIndex].Consumed := TRUE;
			END_IF
			RETURN;
		END_IF

		// Start managing script
		IF NOT _aScripts[nIndex].Started THEN
			_aScripts[nIndex].Started := TRUE;
			_aScripts[nIndex].ActiveCycles := 0;
		END_IF

		// Manage AfterActiveCycle
		IF NOT _aScripts[nIndex].ResultLatched THEN
			_aScripts[nIndex].ActiveCycles := _aScripts[nIndex].ActiveCycles + 1;
			IF (_aScripts[nIndex].AfterActiveCycles = 0)
				OR (_aScripts[nIndex].ActiveCycles >= _aScripts[nIndex].AfterActiveCycles) THEN
			_aScripts[nIndex].ResultLatched := TRUE;
		END_IF
	END_IF

	// Output result if after certain active cycles
	IF _aScripts[nIndex].ResultLatched THEN
		Done := _aScripts[nIndex].Done;
		InVelocity := _aScripts[nIndex].InVelocity;
		Error := _aScripts[nIndex].Error;
		ErrorId := _aScripts[nIndex].ErrorId;
	END_IF
	RETURN;
END_IF
END_FOR
END_METHOD

METHOD M_QueueResult : BOOL
VAR_INPUT
	Operation : E_FakeAxisOperation;
	AfterActiveCycles : UINT;
	Done : BOOL;
	InVelocity : BOOL;
	Error : BOOL;
	ErrorId : UDINT;
END_VAR
M_QueueResult := FALSE;

IF (Operation = E_FakeAxisOperation.None) OR (Done AND Error) THEN
	_bScriptConfigurationError := TRUE;
	RETURN;
END_IF

IF _nScriptCount >= 32 THEN
	_bScriptOverflowed := TRUE;
	RETURN;
END_IF

_nScriptCount := _nScriptCount + 1;
_aScripts[_nScriptCount].Operation := Operation;
_aScripts[_nScriptCount].AfterActiveCycles := AfterActiveCycles;
_aScripts[_nScriptCount].Done := Done;
_aScripts[_nScriptCount].InVelocity := InVelocity;
_aScripts[_nScriptCount].Error := Error;
_aScripts[_nScriptCount].ErrorId := ErrorId;
M_QueueResult := TRUE;
END_METHOD

METHOD PRIVATE M_RecordCall
VAR_INPUT
	Operation : E_FakeAxisOperation;
	OwnerId : T_ResourceOwnerId;
	Accepted : BOOL;
	Execute : BOOL;
	JogForward : BOOL;
	JogBackwards : BOOL;
	Mode : E_JogMode;
	Direction : MC_Direction;
	Position : LREAL;
	Velocity : LREAL;
	Acceleration : LREAL;
	Deceleration : LREAL;
END_VAR
_nCallSequence := _nCallSequence + 1;
IF _nHistoryCount >= 256 THEN
	_bHistoryOverflowed := TRUE;
	RETURN;
END_IF

_nHistoryCount := _nHistoryCount + 1;
_aHistory[_nHistoryCount].Sequence := _nCallSequence;
_aHistory[_nHistoryCount].Cycle := _nCycle;
_aHistory[_nHistoryCount].Operation := Operation;
_aHistory[_nHistoryCount].OwnerId := OwnerId;
_aHistory[_nHistoryCount].Accepted := Accepted;
_aHistory[_nHistoryCount].Execute := Execute;
_aHistory[_nHistoryCount].JogForward := JogForward;
_aHistory[_nHistoryCount].JogBackwards := JogBackwards;
_aHistory[_nHistoryCount].Mode := Mode;
_aHistory[_nHistoryCount].Direction := Direction;
_aHistory[_nHistoryCount].Position := Position;
_aHistory[_nHistoryCount].Velocity := Velocity;
_aHistory[_nHistoryCount].Acceleration := Acceleration;
_aHistory[_nHistoryCount].Deceleration := Deceleration;
END_METHOD

METHOD M_Reset : BOOL
VAR_INPUT
	OwnerId : T_ResourceOwnerId;
	Execute : BOOL;
END_VAR
VAR_OUTPUT
	Done : BOOL;
	Error : BOOL;
	ErrorId : UDINT;
END_VAR
VAR
	bAccepted : BOOL;
END_VAR
bAccepted := M_IsResourceOwner(OwnerId := OwnerId);
M_RecordCall(
	Operation := E_FakeAxisOperation.Reset,
	OwnerId := OwnerId,
	Accepted := bAccepted,
	Execute := Execute,
	JogForward := FALSE,
	JogBackwards := FALSE,
	Mode := E_JogMode.MC_JOGMODE_CONTINOUS,
	Direction := MC_Direction.MC_Positive_Direction,
	Position := 0,
	Velocity := 0,
	Acceleration := 0,
	Deceleration := 0
);

M_Reset := bAccepted;
IF NOT bAccepted THEN
	Done := FALSE;
	Error := FALSE;
	ErrorId := 0;
	RETURN;
END_IF

_bResetActive := Execute;
Done := _bResetDone;
Error := _bResetError;
ErrorId := _nResetErrorId;
END_METHOD

METHOD M_ResetScenario
VAR_INPUT
END_VAR
_ResourceOwnerId := 0;
_bAxisIsDisabled := FALSE;
_bAxisHasJob := FALSE;
_fAxisActualPosition := 0;
_fAxisActualVelocity := 0;
_nCycle := 0;
_nScriptCount := 0;
_bScriptOverflowed := FALSE;
_bScriptConfigurationError := FALSE;
MEMSET(ADR(_aScripts), 0, SIZEOF(_aScripts));
M_ClearCallHistory();

_bJogActive := FALSE;
_bMoveAbsActive := FALSE;
_bMoveVelActive := FALSE;
_bStopActive := FALSE;
_bResetActive := FALSE;
_bHaltActive := FALSE;
_bJogDone := FALSE;
_bJogInVelocity := FALSE;
_bJogError := FALSE;
_nJogErrorId := 0;
_bMoveAbsDone := FALSE;
_bMoveAbsInVelocity := FALSE;
_bMoveAbsError := FALSE;
_nMoveAbsErrorId := 0;
_bMoveVelDone := FALSE;
_bMoveVelInVelocity := FALSE;
_bMoveVelError := FALSE;
_nMoveVelErrorId := 0;
_bStopDone := FALSE;
_bStopInVelocity := FALSE;
_bStopError := FALSE;
_nStopErrorId := 0;
_bResetDone := FALSE;
_bResetInVelocity := FALSE;
_bResetError := FALSE;
_nResetErrorId := 0;
_bHaltDone := FALSE;
_bHaltInVelocity := FALSE;
_bHaltError := FALSE;
_nHaltErrorId := 0;
END_METHOD

METHOD M_SetAxisFeedback
VAR_INPUT
	ActualPosition : LREAL;
	ActualVelocity : LREAL;
END_VAR
_fAxisActualPosition := ActualPosition;
_fAxisActualVelocity := ActualVelocity;
END_METHOD

METHOD M_SetAxisState
VAR_INPUT
	Disabled : BOOL;
	HasJob : BOOL;
END_VAR
_bAxisIsDisabled := Disabled;
_bAxisHasJob := HasJob;
END_METHOD

METHOD M_Stop : BOOL
VAR_INPUT
	OwnerId : T_ResourceOwnerId;
	Execute : BOOL;
	Deceleration : LREAL;
END_VAR
VAR_OUTPUT
	Done : BOOL;
	Error : BOOL;
	ErrorId : UDINT;
END_VAR
VAR
	bAccepted : BOOL;
END_VAR
bAccepted := M_IsResourceOwner(OwnerId := OwnerId);
M_RecordCall(
	Operation := E_FakeAxisOperation.Stop,
	OwnerId := OwnerId,
	Accepted := bAccepted,
	Execute := Execute,
	JogForward := FALSE,
	JogBackwards := FALSE,
	Mode := E_JogMode.MC_JOGMODE_CONTINOUS,
	Direction := MC_Direction.MC_Positive_Direction,
	Position := 0,
	Velocity := 0,
	Acceleration := 0,
	Deceleration := Deceleration
);

M_Stop := bAccepted;
IF NOT bAccepted THEN
	Done := FALSE;
	Error := FALSE;
	ErrorId := 0;
	RETURN;
END_IF

_bStopActive := Execute;
Done := _bStopDone;
Error := _bStopError;
ErrorId := _nStopErrorId;
END_METHOD

PROPERTY ScriptConfigurationError : BOOL
GET
ScriptConfigurationError := _bScriptConfigurationError;
END_GET
END_PROPERTY

PROPERTY ScriptOverflowed : BOOL
GET
ScriptOverflowed := _bScriptOverflowed;
END_GET
END_PROPERTY

END_FUNCTION_BLOCK

// ---- POUs/Test Suites/Infrastructure/FB_UtcClockTests.TcPOU
FUNCTION_BLOCK FB_UtcClockTests EXTENDS TcUnit.FB_TestSuite
VAR
	_Clock : FB_UtcClock;
END_VAR

UtcTimestampHasFixedSortableFormat();

METHOD UtcTimestampHasFixedSortableFormat
VAR
	nIndex : INT;
	sDigit : STRING(1);
	sFirst : STRING(20);
	bDigitsOnly : BOOL;
END_VAR
TEST('UtcTimestampHasFixedSortableFormat');

// Arrange / Act：連續呼叫系統 UTC clock，固定格式應可直接做字典序比較。
_Clock();
sFirst := _Clock.UtcDateTime;
_Clock();

// Assert：YYYYMMDDHHMMSSUUU 共 17 位，且每一位都必須是十進位數字。
bDigitsOnly := LEN(_Clock.UtcDateTime) = 17;
FOR nIndex := 1 TO 17 DO
	sDigit := MID(_Clock.UtcDateTime, 1, nIndex);
	bDigitsOnly := bDigitsOnly AND (FIND('0123456789', sDigit) > 0);
END_FOR
AssertTrue(
	Condition := bDigitsOnly,
	Message := 'UTC timestamp must contain exactly 17 digits.'
);
AssertTrue(
	Condition := _Clock.UtcDateTime >= sFirst,
	Message := 'Consecutive UTC timestamps must not move backwards.'
);

TEST_FINISHED();
END_METHOD

END_FUNCTION_BLOCK

// ---- POUs/Test Suites/PackML/FB_PackMLBaseTests.TcPOU
FUNCTION_BLOCK FB_PackMLBaseTests EXTENDS TcUnit.FB_TestSuite

DefaultLifecycleHonoursBusyHooksAndCompletes();
RejectedCommandFeedbackLatchesUntilRequestFalls();
DisableFreezesStateAndExternalFaultHasPriority();
HoldSuspendStopAndAbortFollowTheStateGuards();

METHOD DefaultLifecycleHonoursBusyHooksAndCompletes
VAR_INST
	Machine : FB_TestPackMLBase;
	Input : ST_PML_Base_In;
	nPhase : UINT;
END_VAR
TEST('DefaultLifecycleHonoursBusyHooksAndCompletes');

CASE nPhase OF
	0:
		// Arrange：第一次掃描由 Undefined 自動完成到 Aborted。
		Machine(PackMLIn := Input);
		AssertTrue(
			Condition := Machine.PackMLOut.eStateCurrent = E_PackMLState.Aborted,
			Message := 'Default Undefined hook must enter Aborted.'
		);
		nPhase := 1;
	1:
		// Act：Clear 後的 transient hook 預設立即完成。
		Input.eCommand := E_PackMLCommand.Clear;
		Input.bCommandChangeRequest := TRUE;
		Machine(PackMLIn := Input);
		AssertTrue(
			Condition := Machine.PackMLOut.eStateCurrent = E_PackMLState.Stopped,
			Message := 'Clear must reach Stopped.'
		);
		nPhase := 2;
	2:
		Input.bCommandChangeRequest := FALSE;
		Machine(PackMLIn := Input);
		nPhase := 3;
	3:
		Input.eCommand := E_PackMLCommand.Reset;
		Input.bCommandChangeRequest := TRUE;
		Machine(PackMLIn := Input);
		AssertTrue(
			Condition := Machine.PackMLOut.eStateCurrent = E_PackMLState.Idle,
			Message := 'Reset must reach Idle.'
		);
		nPhase := 4;
	4:
		Input.bCommandChangeRequest := FALSE;
		Machine(PackMLIn := Input);
		nPhase := 5;
	5:
		// StartingDone=FALSE 驗證 transient state 會跨掃描保持 Busy。
		Input.eCommand := E_PackMLCommand.Start;
		Input.bCommandChangeRequest := TRUE;
		Machine(PackMLIn := Input, StartingDone := FALSE);
		AssertTrue(
			Condition := (Machine.PackMLOut.eStateCurrent = E_PackMLState.Starting)
				AND Machine.bTransitionActive,
			Message := 'Busy Starting must stay active.'
		);
		nPhase := 6;
	6:
		// request 保持 TRUE 時即使 payload 改變，也不能重新消費。
		Input.eCommand := E_PackMLCommand.Abort;
		Machine(PackMLIn := Input, StartingDone := FALSE);
		AssertTrue(
			Condition := Machine.PackMLOut.eStateCurrent = E_PackMLState.Starting,
			Message := 'A held request must not dispatch a new command.'
		);
		nPhase := 7;
	7:
		Input.bCommandChangeRequest := FALSE;
		Machine(PackMLIn := Input, StartingDone := TRUE);
		AssertTrue(
			Condition := Machine.PackMLOut.eStateCurrent = E_PackMLState.Execute,
			Message := 'Done Starting must enter Execute.'
		);
		nPhase := 8;
	8:
		Machine(PackMLIn := Input, ExecuteDone := TRUE);
		AssertTrue(
			Condition := Machine.PackMLOut.eStateCurrent = E_PackMLState.Completing,
			Message := 'Done Execute must enter Completing.'
		);
		nPhase := 9;
	9:
		Machine(PackMLIn := Input, ExecuteDone := TRUE, CompletingDone := TRUE);
		AssertTrue(
			Condition := Machine.PackMLOut.eStateCurrent = E_PackMLState.Complete,
			Message := 'Done Completing must enter Complete.'
		);
		AssertTrue(
			Condition := Machine.FirstScanCalls >= 3,
			Message :=
				'Each entered hook must expose its first scan exactly through the hook argument.'
		);
		nPhase := 0;
		TEST_FINISHED();
END_CASE
END_METHOD

METHOD RejectedCommandFeedbackLatchesUntilRequestFalls
VAR_INST
	Machine : FB_TestPackMLBase;
	Input : ST_PML_Base_In;
	nPhase : UINT;
END_VAR
TEST('RejectedCommandFeedbackLatchesUntilRequestFalls');

CASE nPhase OF
	0:
		Machine(PackMLIn := Input);
		// Aborted
		Input.eCommand := E_PackMLCommand.Start;
		Input.bCommandChangeRequest := TRUE;
		Machine(PackMLIn := Input);
		AssertTrue(
			Condition :=
				Machine.PackMLOut.bCommandRejected
				AND (Machine.PackMLOut.eStateErrorID =
					E_PackMLErrorID.StartNotAllowedFromCurrentState),
			Message := 'Start from Aborted must report the state-specific error.'
		);
		nPhase := 1;
	1:
		// Act：保持 request 為 TRUE，拒絕結果必須鎖存。
		Input.eCommand := E_PackMLCommand.Clear;
		Machine(PackMLIn := Input);
		AssertTrue(
			Condition :=
				Machine.PackMLOut.bCommandRejected
				AND (Machine.PackMLOut.eStateCurrent = E_PackMLState.Aborted),
			Message := 'Held request must preserve rejection and state.'
		);
		nPhase := 2;
	2:
		Input.bCommandChangeRequest := FALSE;
		Machine(PackMLIn := Input);
		AssertFalse(
			Condition := Machine.PackMLOut.bCommandRejected OR Machine.PackMLOut.bCommandAccepted,
			Message := 'Falling edge must clear command feedback.'
		);
		nPhase := 0;
		TEST_FINISHED();
END_CASE
END_METHOD

METHOD DisableFreezesStateAndExternalFaultHasPriority
VAR_INST
	Machine : FB_TestPackMLBase;
	Input : ST_PML_Base_In;
	nPhase : UINT;
END_VAR
TEST('DisableFreezesStateAndExternalFaultHasPriority');

CASE nPhase OF
	0:
		Machine(PackMLIn := Input);
		// Aborted
		Input.eCommand := E_PackMLCommand.Clear;
		Input.bCommandChangeRequest := TRUE;
		Machine(PackMLIn := Input);
		// Stopped
		Input.bCommandChangeRequest := FALSE;
		Machine(PackMLIn := Input);
		nPhase := 1;
	1:
		// Arrange：送 Reset 的同時發生 external fault；Abort 必須優先。
		Input.eCommand := E_PackMLCommand.Reset;
		Input.bCommandChangeRequest := TRUE;
		Machine(PackMLIn := Input, bExternalFault := TRUE);
		AssertTrue(
			Condition := Machine.PackMLOut.eStateCurrent = E_PackMLState.Aborted,
			Message := 'External fault must pre-empt a normal command.'
		);
		nPhase := 2;
	2:
		// Disable 只凍結目前狀態，不可製造 transition activity。
		Machine(PackMLIn := Input, bEnable := FALSE, bExternalFault := FALSE);
		AssertTrue(
			Condition := Machine.PackMLOut.eStateCurrent = E_PackMLState.Aborted,
			Message := 'Disable must preserve state.'
		);
		AssertFalse(
			Condition := Machine.bTransitionActive,
			Message := 'Disable must suppress transition activity.'
		);
		nPhase := 0;
		TEST_FINISHED();
END_CASE
END_METHOD

METHOD HoldSuspendStopAndAbortFollowTheStateGuards
VAR_INST
	Machine : FB_TestPackMLBase;
	Input : ST_PML_Base_In;
	nPhase : UINT;
END_VAR
TEST('HoldSuspendStopAndAbortFollowTheStateGuards');

CASE nPhase OF
	0: Machine(PackMLIn := Input);
	Input.eCommand := E_PackMLCommand.Clear;
	Input.bCommandChangeRequest := TRUE;
	Machine(PackMLIn := Input);
	nPhase := 1;
	1: Input.bCommandChangeRequest := FALSE;
	Machine(PackMLIn := Input);
	Input.eCommand := E_PackMLCommand.Reset;
	Input.bCommandChangeRequest := TRUE;
	Machine(PackMLIn := Input);
	nPhase := 2;
	2: Input.bCommandChangeRequest := FALSE;
	Machine(PackMLIn := Input);
	Input.eCommand := E_PackMLCommand.Start;
	Input.bCommandChangeRequest := TRUE;
	Machine(PackMLIn := Input);
	nPhase := 3;
	3:
		Input.bCommandChangeRequest := FALSE;
		Machine(PackMLIn := Input);
		Input.eCommand := E_PackMLCommand.Hold;
		Input.bCommandChangeRequest := TRUE;
		Machine(PackMLIn := Input);
		AssertTrue(
			Condition := Machine.PackMLOut.eStateCurrent = E_PackMLState.Held,
			Message := 'Hold from Execute must reach Held.'
		);
		nPhase := 4;
	4:
		Input.bCommandChangeRequest := FALSE;
		Machine(PackMLIn := Input);
		Input.eCommand := E_PackMLCommand.Unhold;
		Input.bCommandChangeRequest := TRUE;
		Machine(PackMLIn := Input);
		AssertTrue(
			Condition := Machine.PackMLOut.eStateCurrent = E_PackMLState.Execute,
			Message := 'Unhold from Held must resume Execute.'
		);
		nPhase := 5;
	5:
		Input.bCommandChangeRequest := FALSE;
		Machine(PackMLIn := Input);
		Input.eCommand := E_PackMLCommand.Suspend;
		Input.bCommandChangeRequest := TRUE;
		Machine(PackMLIn := Input);
		AssertTrue(
			Condition := Machine.PackMLOut.eStateCurrent = E_PackMLState.Suspended,
			Message := 'Suspend from Execute must reach Suspended.'
		);
		nPhase := 6;
	6:
		Input.bCommandChangeRequest := FALSE;
		Machine(PackMLIn := Input);
		Input.eCommand := E_PackMLCommand.Unsuspend;
		Input.bCommandChangeRequest := TRUE;
		Machine(PackMLIn := Input);
		AssertTrue(
			Condition := Machine.PackMLOut.eStateCurrent = E_PackMLState.Execute,
			Message := 'Unsuspend must resume Execute.'
		);
		nPhase := 7;
	7:
		Input.bCommandChangeRequest := FALSE;
		Machine(PackMLIn := Input);
		Input.eCommand := E_PackMLCommand.Stop;
		Input.bCommandChangeRequest := TRUE;
		Machine(PackMLIn := Input);
		AssertTrue(
			Condition := Machine.PackMLOut.eStateCurrent = E_PackMLState.Stopped,
			Message := 'Stop from Execute must reach Stopped.'
		);
		nPhase := 8;
	8:
		Input.bCommandChangeRequest := FALSE;
		Machine(PackMLIn := Input);
		Machine(PackMLIn := Input, bExternalFault := TRUE);
		AssertTrue(
			Condition := Machine.PackMLOut.eStateCurrent = E_PackMLState.Aborted,
			Message := 'External fault from Stopped must reach Aborted.'
		);
		nPhase := 0;
		TEST_FINISHED();
END_CASE
END_METHOD

END_FUNCTION_BLOCK

// ---- Fakes/FB_TestPackMLBase.TcPOU
FUNCTION_BLOCK FB_TestPackMLBase EXTENDS FB_PackMLBase
VAR_INPUT
	StartingDone : BOOL := TRUE;
	ExecuteDone : BOOL;
	CompletingDone : BOOL := TRUE;
END_VAR
VAR_OUTPUT
	StartingCalls : UDINT;
	ExecuteCalls : UDINT;
	CompletingCalls : UDINT;
	FirstScanCalls : UDINT;
	StateChangeCalls : UDINT;
	ModeChangeCalls : UDINT;
	LastPreviousState : E_PackMLState;
	LastNewState : E_PackMLState;
END_VAR

SUPER^();

METHOD PROTECTED H_OnStarting : E_PackMLHookResult
VAR_INPUT
	bFirstScan : BOOL;
END_VAR
StartingCalls := StartingCalls + 1;
IF bFirstScan THEN
	FirstScanCalls := FirstScanCalls + 1;
END_IF
IF StartingDone THEN
	H_OnStarting := E_PackMLHookResult.Done;
ELSE
	H_OnStarting := E_PackMLHookResult.Busy;
END_IF
END_METHOD

METHOD PROTECTED H_OnExecute : E_PackMLHookResult
VAR_INPUT
	bFirstScan : BOOL;
END_VAR
ExecuteCalls := ExecuteCalls + 1;
IF bFirstScan THEN
	FirstScanCalls := FirstScanCalls + 1;
END_IF
IF ExecuteDone THEN
	H_OnExecute := E_PackMLHookResult.Done;
ELSE
	H_OnExecute := E_PackMLHookResult.Busy;
END_IF
END_METHOD

METHOD PROTECTED H_OnCompleting : E_PackMLHookResult
VAR_INPUT
	bFirstScan : BOOL;
END_VAR
CompletingCalls := CompletingCalls + 1;
IF bFirstScan THEN
	FirstScanCalls := FirstScanCalls + 1;
END_IF
IF CompletingDone THEN
	H_OnCompleting := E_PackMLHookResult.Done;
ELSE
	H_OnCompleting := E_PackMLHookResult.Busy;
END_IF
END_METHOD

METHOD PROTECTED H_OnStateChanged
VAR_INPUT
	ePreviousState : E_PackMLState;
	eNewState : E_PackMLState;
END_VAR
StateChangeCalls := StateChangeCalls + 1;
LastPreviousState := ePreviousState;
LastNewState := eNewState;
END_METHOD

METHOD PROTECTED H_OnModeChanged
VAR_INPUT
	ePreviousMode : T_PackMLMode;
	eNewMode : T_PackMLMode;
END_VAR
ModeChangeCalls := ModeChangeCalls + 1;
END_METHOD

METHOD PUBLIC M_TestRequestCommand : BOOL
VAR_INPUT
	Command : E_PackMLCommand;
END_VAR
M_TestRequestCommand := RequestCommand(eTargetCmd := Command);
END_METHOD

END_FUNCTION_BLOCK

// ---- POUs/Test Suites/PackML/FB_PackMLModeSetTests.TcPOU
FUNCTION_BLOCK FB_PackMLModeSetTests EXTENDS TcUnit.FB_TestSuite
VAR
	_ModeSet : FB_TestPackMLModeSet;
END_VAR

SupportedModesAreExplicit();
ManualModeUsesTheSafetyWhitelist();
ManualAndProductionStateMatricesDiffer();

METHOD SupportedModesAreExplicit
TEST('SupportedModesAreExplicit');

// Assert：只有 Manual 與 Production 是公開支援模式。
AssertTrue(
	Condition := _ModeSet.M_IsModeAllowed(Mode := E_PackMLMode.Manual),
	Message := 'Manual mode must be supported.'
);
AssertTrue(
	Condition := _ModeSet.M_IsModeAllowed(Mode := E_PackMLMode.Production),
	Message := 'Production mode must be supported.'
);
AssertFalse(
	Condition := _ModeSet.M_IsModeAllowed(Mode := E_PackMLMode.Unknown),
	Message := 'Unknown mode must be rejected.'
);

TEST_FINISHED();
END_METHOD

METHOD ManualModeUsesTheSafetyWhitelist
TEST('ManualModeUsesTheSafetyWhitelist');

// Arrange / Act / Assert：Manual 只允許 reset/start/stop/abort/clear。
AssertTrue(
	Condition := _ModeSet.M_IsCommandAllowed(
		Command := E_PackMLCommand.Reset,
		Mode := E_PackMLMode.Manual
	),
	Message := 'Manual Reset must be allowed.'
);
AssertTrue(
	Condition := _ModeSet.M_IsCommandAllowed(
		Command := E_PackMLCommand.Start,
		Mode := E_PackMLMode.Manual
	),
	Message := 'Manual Start must be allowed.'
);
AssertTrue(
	Condition := _ModeSet.M_IsCommandAllowed(
		Command := E_PackMLCommand.Stop,
		Mode := E_PackMLMode.Manual
	),
	Message := 'Manual Stop must be allowed.'
);
AssertTrue(
	Condition := _ModeSet.M_IsCommandAllowed(
		Command := E_PackMLCommand.Abort,
		Mode := E_PackMLMode.Manual
	),
	Message := 'Manual Abort must be allowed.'
);
AssertTrue(
	Condition := _ModeSet.M_IsCommandAllowed(
		Command := E_PackMLCommand.Clear,
		Mode := E_PackMLMode.Manual
	),
	Message := 'Manual Clear must be allowed.'
);
AssertFalse(
	Condition := _ModeSet.M_IsCommandAllowed(
		Command := E_PackMLCommand.Hold,
		Mode := E_PackMLMode.Manual
	),
	Message := 'Manual Hold must be rejected.'
);
AssertFalse(
	Condition := _ModeSet.M_IsCommandAllowed(
		Command := E_PackMLCommand.Unhold,
		Mode := E_PackMLMode.Manual
	),
	Message := 'Manual Unhold must be rejected.'
);
AssertFalse(
	Condition := _ModeSet.M_IsCommandAllowed(
		Command := E_PackMLCommand.Suspend,
		Mode := E_PackMLMode.Manual
	),
	Message := 'Manual Suspend must be rejected.'
);
AssertFalse(
	Condition := _ModeSet.M_IsCommandAllowed(
		Command := E_PackMLCommand.Unsuspend,
		Mode := E_PackMLMode.Manual
	),
	Message := 'Manual Unsuspend must be rejected.'
);

TEST_FINISHED();
END_METHOD

METHOD ManualAndProductionStateMatricesDiffer
TEST('ManualAndProductionStateMatricesDiffer');

// Manual 允許核心操作狀態，但不允許 Held、Suspended、Complete。
AssertTrue(
	Condition := _ModeSet.M_IsStateAllowed(
		Mode := E_PackMLMode.Manual,
		State := E_PackMLState.Idle
	),
	Message := 'Manual Idle must be supported.'
);
AssertTrue(
	Condition := _ModeSet.M_IsStateAllowed(
		Mode := E_PackMLMode.Manual,
		State := E_PackMLState.Execute
	),
	Message := 'Manual Execute must be supported.'
);
AssertFalse(
	Condition := _ModeSet.M_IsStateAllowed(
		Mode := E_PackMLMode.Manual,
		State := E_PackMLState.Held
	),
	Message := 'Manual Held must be rejected.'
);
AssertFalse(
	Condition := _ModeSet.M_IsStateAllowed(
		Mode := E_PackMLMode.Manual,
		State := E_PackMLState.Suspended
	),
	Message := 'Manual Suspended must be rejected.'
);
AssertFalse(
	Condition := _ModeSet.M_IsStateAllowed(
		Mode := E_PackMLMode.Manual,
		State := E_PackMLState.Complete
	),
	Message := 'Manual Complete must be rejected.'
);

// Production 接受完整 PackML state surface。
AssertTrue(
	Condition := _ModeSet.M_IsStateAllowed(
		Mode := E_PackMLMode.Production,
		State := E_PackMLState.Held
	),
	Message := 'Production Held must be supported.'
);
AssertTrue(
	Condition := _ModeSet.M_IsCommandAllowed(
		Command := E_PackMLCommand.Suspend,
		Mode := E_PackMLMode.Production
	),
	Message := 'Production Suspend must be supported.'
);

TEST_FINISHED();
END_METHOD

END_FUNCTION_BLOCK

// ---- Fakes/FB_TestPackMLModeSet.TcPOU
FUNCTION_BLOCK FB_TestPackMLModeSet EXTENDS FB_PackMLModeSet

SUPER^();

METHOD PUBLIC M_IsCommandAllowed : BOOL
VAR_INPUT
	Command : E_PackMLCommand;
	Mode : T_PackMLMode;
END_VAR
M_IsCommandAllowed := H_IsCommandAllowedByMode(
	eRequestedCommand := Command,
	eActiveMode := Mode
);
END_METHOD

METHOD PUBLIC M_IsModeAllowed : BOOL
VAR_INPUT
	Mode : T_PackMLMode;
END_VAR
M_IsModeAllowed := H_IsModeSupported(eRequestedMode := Mode);
END_METHOD

METHOD PUBLIC M_IsStateAllowed : BOOL
VAR_INPUT
	Mode : T_PackMLMode;
	State : E_PackMLState;
END_VAR
M_IsStateAllowed := H_IsStateSupportedByMode(
	eRequestedMode := Mode,
	eCurrentState := State
);
END_METHOD

END_FUNCTION_BLOCK

// ---- POUs/Test Suites/Service/FB_ServiceBaseTests.TcPOU
FUNCTION_BLOCK FB_ServiceBaseTests EXTENDS TcUnit.FB_TestSuite
VAR
	// Keep the Service instance at Test Suite scope so its state persists across test phases.
	TestService : FB_TestableServiceBase;
END_VAR

StartCommandIsRejectedWhileStopped();
ErrorListPreservesFirstOccurrenceAndCapacity();
DataListSupportsUpsertClearAndOverflow();

METHOD StartCommandIsRejectedWhileStopped
VAR_INST
	Ctrl : ST_ServiceCtrl;
	Context : ST_ServiceContext;
	nPhase : UINT;
END_VAR
TEST('StartCommandIsRejectedWhileStopped');

CASE nPhase OF
	0:
		// Initial cyclic update leaves Undefined through the normal ServiceBase path.
		TestService(
			Ctrl := Ctrl,
			Context := Context,
			ServiceId := 1);

		AssertTrue(
			Condition := TestService.Status.PackMLOut.eStateCurrent = E_PackMLState.Aborted,
			Message := 'Initial Service update must reach Aborted.');
		AssertTrue(
			Condition := TestService.Status.CompletionBehavior =
				E_ServiceCompletionBehavior.Unknown,
			Message :=
				'The test Service must publish its configured Unknown completion behavior.');
		nPhase := 1;

	1:
		// Clear is valid from Aborted and establishes Stopped through a public command.
		Ctrl.RequestId := 1001;
		Ctrl.PackMLIn.eCommand := E_PackMLCommand.Clear;
		Ctrl.PackMLIn.bCommandChangeRequest := TRUE;
		TestService(
			Ctrl := Ctrl,
			Context := Context,
			ServiceId := 1);

		AssertTrue(
			Condition := TestService.Status.PackMLOut.eStateCurrent = E_PackMLState.Stopped,
			Message := 'Valid Clear from Aborted must establish Stopped.');
		AssertTrue(
			Condition := TestService.Status.PackMLOut.bCommandAccepted
				AND NOT TestService.Status.PackMLOut.bCommandRejected,
			Message := 'Clear must be accepted while establishing the test state.');
		AssertTrue(
			Condition := TestService.Status.ResponseId = 1001,
			Message := 'Service must acknowledge the Clear request.');
		nPhase := 2;

	2:
		// Withdraw Clear so the next command creates a new request edge.
		Ctrl.PackMLIn.bCommandChangeRequest := FALSE;
		TestService(
			Ctrl := Ctrl,
			Context := Context,
			ServiceId := 1);

		AssertTrue(
			Condition := (TestService.Status.PackMLOut.eStateCurrent = E_PackMLState.Stopped)
				AND NOT TestService.Status.PackMLOut.bCommandAccepted
				AND NOT TestService.Status.PackMLOut.bCommandRejected
				AND (TestService.Status.PackMLOut.eStateErrorID = E_PackMLErrorID.NoError),
			Message := 'Withdrawing Clear must leave a clean Stopped command interface.');
		nPhase := 3;

	3:
		// Start is only valid from Idle, so Stopped must reject it without transitioning.
		Ctrl.RequestId := 1002;
		Ctrl.PackMLIn.eCommand := E_PackMLCommand.Start;
		Ctrl.PackMLIn.bCommandChangeRequest := TRUE;
		TestService(
			Ctrl := Ctrl,
			Context := Context,
			ServiceId := 1);

		AssertTrue(
			Condition := TestService.Status.PackMLOut.eStateCurrent = E_PackMLState.Stopped,
			Message := 'Rejected Start must not leave Stopped.');
		AssertTrue(
			Condition := TestService.Status.PackMLOut.bCommandRejected
				AND NOT TestService.Status.PackMLOut.bCommandAccepted,
			Message := 'Start must be rejected while the Service is Stopped.');
		AssertTrue(
			Condition := TestService.Status.PackMLOut.eStateErrorID =
				E_PackMLErrorID.StartNotAllowedFromCurrentState,
			Message := 'Rejected Start must report the state-specific PackML ErrorID.');
		AssertTrue(
			Condition := TestService.Status.ResponseId = 1002,
			Message := 'Service must acknowledge the rejected Start request.');
		nPhase := 4;

	4:
		// A held request is already consumed; changing its payload must not execute Reset.
		Ctrl.RequestId := 1003;
		Ctrl.PackMLIn.eCommand := E_PackMLCommand.Reset;
		TestService(
			Ctrl := Ctrl,
			Context := Context,
			ServiceId := 1);

		AssertTrue(
			Condition := TestService.Status.PackMLOut.eStateCurrent = E_PackMLState.Stopped,
			Message := 'A command request held TRUE must not be processed again.');
		AssertTrue(
			Condition := TestService.Status.PackMLOut.bCommandRejected
				AND (TestService.Status.PackMLOut.eStateErrorID =
					E_PackMLErrorID.StartNotAllowedFromCurrentState),
			Message :=
				'Rejected Start feedback must stay latched while the request remains TRUE.');
		AssertTrue(
			Condition := TestService.Status.ResponseId = 1002,
			Message := 'Changing request data without a falling edge must not update ResponseId.');
		nPhase := 5;

	5:
		// The request falling edge clears rejection feedback and arms the next command.
		Ctrl.PackMLIn.bCommandChangeRequest := FALSE;
		TestService(
			Ctrl := Ctrl,
			Context := Context,
			ServiceId := 1);

		AssertTrue(
			Condition := (TestService.Status.PackMLOut.eStateCurrent = E_PackMLState.Stopped)
				AND NOT TestService.Status.PackMLOut.bCommandAccepted
				AND NOT TestService.Status.PackMLOut.bCommandRejected
				AND (TestService.Status.PackMLOut.eStateErrorID = E_PackMLErrorID.NoError),
			Message := 'The request falling edge must clear rejected command feedback.');
		nPhase := 6;

	6:
		// A fresh Reset request proves rejection did not block later valid commands.
		Ctrl.RequestId := 1004;
		Ctrl.PackMLIn.eCommand := E_PackMLCommand.Reset;
		Ctrl.PackMLIn.bCommandChangeRequest := TRUE;
		TestService(
			Ctrl := Ctrl,
			Context := Context,
			ServiceId := 1);

		AssertTrue(
			Condition := TestService.Status.PackMLOut.eStateCurrent = E_PackMLState.Idle,
			Message := 'Fresh Reset from Stopped must remain operable after a rejected Start.');
		AssertTrue(
			Condition := TestService.Status.PackMLOut.bCommandAccepted
				AND NOT TestService.Status.PackMLOut.bCommandRejected
				AND (TestService.Status.PackMLOut.eStateErrorID = E_PackMLErrorID.NoError),
			Message := 'Fresh Reset must be accepted after rejection feedback is cleared.');
		AssertTrue(
			Condition := TestService.Status.ResponseId = 1004,
			Message := 'Service must acknowledge the fresh Reset request.');
		AssertTrue(
			Condition := TestService.Status.CompletionBehavior =
				E_ServiceCompletionBehavior.Unknown,
			Message := 'Completion behavior must remain stable across PackML state transitions.');

		nPhase := 0;
		TEST_FINISHED();
END_CASE
END_METHOD

METHOD ErrorListPreservesFirstOccurrenceAndCapacity
VAR_INST
	Service : FB_TestableServiceBase;
	Ctrl : ST_ServiceCtrl;
	Context : ST_ServiceContext;
	bInitialized : BOOL;
END_VAR
VAR
	nIndex : UINT;
	bAccepted : BOOL;
END_VAR
TEST('ErrorListPreservesFirstOccurrenceAndCapacity');

IF NOT bInitialized THEN
	// Arrange：先綁定持久 Context，確保錯誤 metadata 可安全取用。
	Context.ModuleId := 41;
	Context.UtcDateTime := '20260921120000000';
	Service(Ctrl := Ctrl, Context := Context, ServiceId := 7);
	Service.M_TestClearErrors();

	// Act：第一筆成立；同 MainErrorId 在同一輪不得重複新增。
	AssertTrue(
		Condition := Service.M_TestAddError(
			MainErrorId := 100,
			SourceErrorId := 5,
			Message := 'first'
		),
		Message := 'First error must be accepted.'
	);
	AssertFalse(
		Condition := Service.M_TestAddError(
			MainErrorId := 100,
			SourceErrorId := 9,
			Message := 'duplicate'
		),
		Message := 'Duplicate MainErrorId must be rejected.'
	);
	FOR nIndex := 2 TO Param_Config.MaxServiceError DO
		bAccepted := Service.M_TestAddError(
			MainErrorId := 99 + UINT_TO_UDINT(nIndex),
			SourceErrorId := 0,
			Message := 'fill'
		);
	END_FOR
	AssertFalse(
		Condition := Service.M_TestAddError(
			MainErrorId := 999,
			SourceErrorId := 0,
			Message := 'overflow'
		),
		Message := 'The first ten errors must be preserved at capacity.'
	);

	// Assert：framework 補上的 Module、Service、時間與 lifecycle 欄位正確。
	AssertTrue(
		Condition := (Service.Status.ErrorList[1].ModuleId = 41)
			AND (Service.Status.ErrorList[1].ServiceId = 7),
		Message := 'Error identity must include Module and Service.'
	);
	AssertTrue(
		Condition :=
			(Service.Status.ErrorList[1].Message = 'first')
			AND (Service.Status.ErrorList[1].SourceErrorId = 5),
		Message := 'Duplicate submission must not replace the first snapshot.'
	);
	AssertTrue(
		Condition := Service.Status.ErrorList[1].Active
			AND NOT Service.Status.ErrorList[1].Acknowledged,
		Message := 'A new Service error must be active and unacknowledged.'
	);
	bInitialized := TRUE;
END_IF

TEST_FINISHED();
END_METHOD

METHOD DataListSupportsUpsertClearAndOverflow
VAR_INST
	Service : FB_TestableServiceBase;
	Ctrl : ST_ServiceCtrl;
	Context : ST_ServiceContext;
	bInitialized : BOOL;
END_VAR
VAR
	nIndex : UINT;
	bAccepted : BOOL;
END_VAR
TEST('DataListSupportsUpsertClearAndOverflow');

IF NOT bInitialized THEN
	Service(Ctrl := Ctrl, Context := Context, ServiceId := 8);
	Service.M_TestClearAllData();

	// Arrange / Act：相同 DataId 是更新，不增加 Count。
	AssertFalse(
		Condition := Service.M_TestUpdateData(
			DataId := 0,
			Name := 'invalid',
			DataType := E_DescriptorType.Integer_32bit,
			Unit := '',
			Value := '0'
		),
		Message := 'DataId zero must be rejected.'
	);
	AssertTrue(
		Condition := Service.M_TestUpdateData(
			DataId := 1,
			Name := 'speed',
			DataType := E_DescriptorType.Float_64bit,
			Unit := 'rpm',
			Value := '10'
		),
		Message := 'First data value must be accepted.'
	);
	AssertTrue(
		Condition := Service.M_TestUpdateData(
			DataId := 1,
			Name := 'speed',
			DataType := E_DescriptorType.Float_64bit,
			Unit := 'rpm',
			Value := '20'
		),
		Message := 'Existing data must be updated.'
	);
	AssertTrue(
		Condition := (Service.Status.Data.Count = 1)
			AND (Service.Status.Data.DataList[1].Value = '20'),
		Message := 'Upsert must retain one entry with the latest value.'
	);

	// Act：清除會釋放容量並重設 overflow。
	AssertTrue(
		Condition := Service.M_TestClearData(DataId := 1),
		Message := 'Existing data must be removable.'
	);
	AssertFalse(
		Condition := Service.M_TestClearData(DataId := 1),
		Message := 'Clearing a missing data ID must report false.'
	);
	FOR nIndex := 1 TO Param_Config.MaxServiceData DO
		bAccepted := Service.M_TestUpdateData(
			DataId := UINT_TO_UDINT(nIndex),
			Name := 'fill',
			DataType := E_DescriptorType.Integer_32bit,
			Unit := '',
			Value := '1'
		);
	END_FOR
	AssertFalse(
		Condition := Service.M_TestUpdateData(
			DataId := 999,
			Name := 'overflow',
			DataType := E_DescriptorType.Integer_32bit,
			Unit := '',
			Value := '1'
		),
		Message := 'Data beyond capacity must be rejected.'
	);
	AssertTrue(
		Condition := Service.Status.Data.Overflow
			AND (Service.Status.Data.Count = Param_Config.MaxServiceData),
		Message := 'Capacity rejection must set Overflow without changing Count.'
	);
	bInitialized := TRUE;
END_IF

TEST_FINISHED();
END_METHOD

END_FUNCTION_BLOCK

// ---- Fakes/FB_TestableServiceBase.TcPOU
FUNCTION_BLOCK FB_TestableServiceBase EXTENDS FB_ServiceBase
VAR_INPUT
	TestExecuteSubState : UDINT;
	TestExecuteSubStateName : STRING(80);
	StartingBusyScans : UINT;
	CompleteExecute : BOOL;
END_VAR
VAR
	_StartingBusyScanCount : UINT;
END_VAR

M_UpdateService(CompletionBehavior := E_ServiceCompletionBehavior.Unknown);

METHOD PROTECTED H_GetExecuteSubState : UDINT
H_GetExecuteSubState := TestExecuteSubState;
END_METHOD

METHOD PROTECTED H_GetExecuteSubStateName : STRING(80)
H_GetExecuteSubStateName := TestExecuteSubStateName;
END_METHOD

METHOD PROTECTED H_OnExecute : E_PackMLHookResult
VAR_INPUT
	bFirstScan : BOOL;
END_VAR
IF CompleteExecute THEN
	H_OnExecute := E_PackMLHookResult.Done;
ELSE
	H_OnExecute := E_PackMLHookResult.Busy;
END_IF
END_METHOD

METHOD PROTECTED H_OnStarting : E_PackMLHookResult
VAR_INPUT
	bFirstScan : BOOL;
END_VAR
IF bFirstScan THEN
	_StartingBusyScanCount := 0;
END_IF

IF _StartingBusyScanCount < StartingBusyScans THEN
	_StartingBusyScanCount := _StartingBusyScanCount + 1;
	H_OnStarting := E_PackMLHookResult.Busy;
ELSE
	H_OnStarting := E_PackMLHookResult.Done;
END_IF
END_METHOD

METHOD PUBLIC M_TestAddError : BOOL
VAR_INPUT
	MainErrorId : UDINT;
	SourceErrorId : UDINT;
	Message : STRING;
END_VAR
M_TestAddError := M_AddError(
	MainErrorId := MainErrorId,
	SourceErrorId := SourceErrorId,
	Message := Message
);
END_METHOD

METHOD PUBLIC M_TestClearErrors : BOOL
M_TestClearErrors := M_ClearAllError();
END_METHOD

METHOD PUBLIC M_TestUpdateData : BOOL
VAR_INPUT
	DataId : UDINT;
	Name : STRING(30);
	DataType : E_DescriptorType;
	Unit : STRING(10);
	Value : STRING(80);
END_VAR
M_TestUpdateData := M_UpdateData(
	DataId := DataId,
	Name := Name,
	DataType := DataType,
	Unit := Unit,
	Value := Value
);
END_METHOD

METHOD PUBLIC M_TestClearData : BOOL
VAR_INPUT
	DataId : UDINT;
END_VAR
M_TestClearData := M_ClearData(DataId := DataId);
END_METHOD

METHOD PUBLIC M_TestClearAllData
M_ClearAllData();
END_METHOD

END_FUNCTION_BLOCK

// ---- POUs/Test Suites/Service/FB_ServiceExecuteSubStateTests.TcPOU
FUNCTION_BLOCK FB_ServiceExecuteSubStateTests EXTENDS TcUnit.FB_TestSuite
VAR
	TimelineService : FB_TestableServiceBase;
	OverflowService : FB_TestableServiceBase;
	CarryoverService : FB_TestableCarryoverSubStateService;
	SnapshotCoordinator : FB_ServiceCoordinator;
END_VAR

SecondRunDoesNotRecordCarryoverFinish();
TimelineTracksTransitionsAndClearsOnStarting();
OverflowPreservesFirstThirtyRecords();
CoordinatorSnapshotUsesCurrentStepOnly();

METHOD CoordinatorSnapshotUsesCurrentStepOnly
VAR_INST
	UpperCtrl : ST_ServiceCtrl;
	EffectiveCtrl : ST_ServiceCtrl;
	UpperParam : UDINT;
	EffectiveParam : UDINT;
	Status : ST_ServiceStatus;
	Snapshot : ST_ServiceExecutionSnapshot;
	bInitialized : BOOL;
END_VAR
VAR
	bOk : BOOL;
END_VAR
TEST('CoordinatorSnapshotUsesCurrentStepOnly');

IF NOT bInitialized THEN
	bOk := SnapshotCoordinator.M_BeginRegistration();
	bOk := bOk AND SnapshotCoordinator.M_Register(
		ServiceId := 17,
		AllowCompositeCall := FALSE,
		UpperParam := UpperParam,
		EffectiveParam := EffectiveParam,
		UpperCtrl := UpperCtrl,
		EffectiveCtrl := EffectiveCtrl,
		Status := Status);
	bOk := bOk AND SnapshotCoordinator.M_Seal();
	bInitialized := TRUE;
ELSE
	bOk := SnapshotCoordinator.Ready;
END_IF

Status.ServiceId := 17;
Status.PackMLOut.eStateCurrent := E_PackMLState.Execute;
Status.ExecuteSubState.CurrentStep := 42;
Status.ExecuteSubState.RecordCount := 1;
Status.ExecuteSubState.Records[1].Step := 7;
SnapshotCoordinator.M_ObserveCycle();
bOk := bOk AND SnapshotCoordinator.M_GetServiceSnapshotById(
	ServiceId := 17,
	Snapshot => Snapshot
);

AssertTrue(Condition := bOk AND Snapshot.Valid AND (Snapshot.ExecuteSubState = 42),
	Message := 'Coordinator snapshots must copy only ExecuteSubState.CurrentStep.');
TEST_FINISHED();
END_METHOD

METHOD OverflowPreservesFirstThirtyRecords
VAR_INST
	Ctrl : ST_ServiceCtrl;
	Context : ST_ServiceContext;
	nPhase : UINT;
	NextState : UDINT := 1;
END_VAR
TEST('OverflowPreservesFirstThirtyRecords');

CASE nPhase OF
	0:
		OverflowService(Ctrl := Ctrl, Context := Context, ServiceId := 2,
			TestExecuteSubState := 0, TestExecuteSubStateName := 'Overflow');
		nPhase := 1;
	1:
		Ctrl.PackMLIn.eCommand := E_PackMLCommand.Clear;
		Ctrl.PackMLIn.bCommandChangeRequest := TRUE;
		OverflowService(Ctrl := Ctrl, Context := Context, ServiceId := 2);
		nPhase := 2;
	2:
		Ctrl.PackMLIn.bCommandChangeRequest := FALSE;
		OverflowService(Ctrl := Ctrl, Context := Context, ServiceId := 2);
		nPhase := 3;
	3:
		Ctrl.PackMLIn.eCommand := E_PackMLCommand.Reset;
		Ctrl.PackMLIn.bCommandChangeRequest := TRUE;
		OverflowService(Ctrl := Ctrl, Context := Context, ServiceId := 2);
		nPhase := 4;
	4:
		Ctrl.PackMLIn.bCommandChangeRequest := FALSE;
		OverflowService(Ctrl := Ctrl, Context := Context, ServiceId := 2);
		nPhase := 5;
	5:
		Context.UtcDateTime := '20260916100000000';
		Ctrl.PackMLIn.eCommand := E_PackMLCommand.Start;
		Ctrl.PackMLIn.bCommandChangeRequest := TRUE;
		OverflowService(Ctrl := Ctrl, Context := Context, ServiceId := 2,
			TestExecuteSubState := 1);
		nPhase := 6;
	6:
		Ctrl.PackMLIn.bCommandChangeRequest := FALSE;
		IF NextState <= 31 THEN
			OverflowService(Ctrl := Ctrl, Context := Context, ServiceId := 2,
				TestExecuteSubState := NextState);
			NextState := NextState + 1;
		ELSE
			nPhase := 7;
		END_IF
	7:
		AssertTrue(Condition := (OverflowService.Status.ExecuteSubState.CurrentStep = 31)
				AND (OverflowService.Status.ExecuteSubState.RecordCount =
					Param_Config.MaxExecuteSubStateRecords)
				AND OverflowService.Status.ExecuteSubState.Overflow,
			Message :=
				'The thirty-first transition must set Overflow while retaining the current state.');
		AssertTrue(Condition := (OverflowService.Status.ExecuteSubState.Records[1].Step = 1)
				AND (OverflowService.Status.ExecuteSubState.Records[30].Step = 30)
				AND (OverflowService.Status.ExecuteSubState.Records[30].EndTimestamp <> ''),
			Message := 'Overflow must preserve the first thirty complete record slots.');
		Context.UtcDateTime := '20260916100100000';
		Ctrl.PackMLIn.eCommand := E_PackMLCommand.Stop;
		Ctrl.PackMLIn.bCommandChangeRequest := TRUE;
		OverflowService(Ctrl := Ctrl, Context := Context, ServiceId := 2);
		nPhase := 8;
	8:
		Ctrl.PackMLIn.bCommandChangeRequest := FALSE;
		OverflowService(Ctrl := Ctrl, Context := Context, ServiceId := 2);
		nPhase := 9;
	9:
		Ctrl.PackMLIn.eCommand := E_PackMLCommand.Reset;
		Ctrl.PackMLIn.bCommandChangeRequest := TRUE;
		OverflowService(Ctrl := Ctrl, Context := Context, ServiceId := 2);
		nPhase := 10;
	10:
		Ctrl.PackMLIn.bCommandChangeRequest := FALSE;
		OverflowService(Ctrl := Ctrl, Context := Context, ServiceId := 2);
		nPhase := 11;
	11:
		Context.UtcDateTime := '20260916100200000';
		Ctrl.PackMLIn.eCommand := E_PackMLCommand.Start;
		Ctrl.PackMLIn.bCommandChangeRequest := TRUE;
		OverflowService(Ctrl := Ctrl, Context := Context, ServiceId := 2,
			TestExecuteSubState := 99);
		AssertTrue(Condition := (OverflowService.Status.ExecuteSubState.CurrentStep = 0)
				AND (OverflowService.Status.ExecuteSubState.RecordCount = 0)
				AND NOT OverflowService.Status.ExecuteSubState.Overflow
				AND (OverflowService.Status.ExecuteSubState.Records[1].Step = 0),
			Message :=
				'The next Starting must clear Count, Overflow, and every old record before sampling.');
		nPhase := 12;
	12:
		Context.UtcDateTime := '20260916100200001';
		Ctrl.PackMLIn.bCommandChangeRequest := FALSE;
		OverflowService(Ctrl := Ctrl, Context := Context, ServiceId := 2,
			TestExecuteSubState := 99);
		AssertTrue(Condition := (OverflowService.Status.ExecuteSubState.CurrentStep = 99)
				AND (OverflowService.Status.ExecuteSubState.RecordCount = 1)
				AND NOT OverflowService.Status.ExecuteSubState.Overflow
				AND (OverflowService.Status.ExecuteSubState.Records[1].Step = 99)
				AND (OverflowService.Status.ExecuteSubState.Records[2].Step = 0),
			Message :=
				'The first evaluated Execute action must start the new timeline after clearing.');
		NextState := 1;
		nPhase := 0;
		TEST_FINISHED();
END_CASE
END_METHOD

METHOD SecondRunDoesNotRecordCarryoverFinish
VAR_INST
	Ctrl : ST_ServiceCtrl;
	Context : ST_ServiceContext;
	nPhase : UINT;
END_VAR
TEST('SecondRunDoesNotRecordCarryoverFinish');

CASE nPhase OF
	0:
		CarryoverService(Ctrl := Ctrl, Context := Context, ServiceId := 3);
		nPhase := 1;
	1:
		Ctrl.PackMLIn.eCommand := E_PackMLCommand.Clear;
		Ctrl.PackMLIn.bCommandChangeRequest := TRUE;
		CarryoverService(Ctrl := Ctrl, Context := Context, ServiceId := 3);
		nPhase := 2;
	2:
		Ctrl.PackMLIn.bCommandChangeRequest := FALSE;
		CarryoverService(Ctrl := Ctrl, Context := Context, ServiceId := 3);
		nPhase := 3;
	3:
		Ctrl.PackMLIn.eCommand := E_PackMLCommand.Reset;
		Ctrl.PackMLIn.bCommandChangeRequest := TRUE;
		CarryoverService(Ctrl := Ctrl, Context := Context, ServiceId := 3);
		nPhase := 4;
	4:
		Ctrl.PackMLIn.bCommandChangeRequest := FALSE;
		CarryoverService(Ctrl := Ctrl, Context := Context, ServiceId := 3);
		nPhase := 5;
	5:
		Context.UtcDateTime := '20260916110000000';
		Ctrl.PackMLIn.eCommand := E_PackMLCommand.Start;
		Ctrl.PackMLIn.bCommandChangeRequest := TRUE;
		CarryoverService(Ctrl := Ctrl, Context := Context, ServiceId := 3);
		AssertTrue(
			Condition := (CarryoverService.Status.PackMLOut.eStateCurrent = E_PackMLState.Execute)
				AND (CarryoverService.Status.ExecuteSubState.CurrentStep = 0)
				AND (CarryoverService.Status.ExecuteSubState.RecordCount = 0),
			Message :=
				'Starting-to-Execute transition must not record the previous Finish substate.');
		nPhase := 6;
	6:
		Context.UtcDateTime := '20260916110000001';
		Ctrl.PackMLIn.bCommandChangeRequest := FALSE;
		CarryoverService(Ctrl := Ctrl, Context := Context, ServiceId := 3);
		AssertTrue(
			Condition := (CarryoverService.Status.ExecuteSubState.CurrentStep = 1)
				AND (CarryoverService.Status.ExecuteSubState.RecordCount = 1)
				AND (CarryoverService.Status.ExecuteSubState.Records[1].Step = 1)
				AND (CarryoverService.Status.ExecuteSubState.Records[1].Name = 'LiftReady')
				AND (CarryoverService.Status.ExecuteSubState.Records[2].Step = 0),
			Message := 'First evaluated Execute scan must start directly with LiftReady.');
		nPhase := 0;
		TEST_FINISHED();
END_CASE
END_METHOD

METHOD TimelineTracksTransitionsAndClearsOnStarting
VAR_INST
	Ctrl : ST_ServiceCtrl;
	Context : ST_ServiceContext;
	nPhase : UINT;
END_VAR
TEST('TimelineTracksTransitionsAndClearsOnStarting');

CASE nPhase OF
	0:
		TimelineService(Ctrl := Ctrl, Context := Context, ServiceId := 1,
			TestExecuteSubState := 0, TestExecuteSubStateName := '',
			StartingBusyScans := 0, CompleteExecute := FALSE);
		nPhase := 1;

	1:
		Ctrl.PackMLIn.eCommand := E_PackMLCommand.Clear;
		Ctrl.PackMLIn.bCommandChangeRequest := TRUE;
		TimelineService(Ctrl := Ctrl, Context := Context, ServiceId := 1);
		nPhase := 2;

	2:
		Ctrl.PackMLIn.bCommandChangeRequest := FALSE;
		TimelineService(Ctrl := Ctrl, Context := Context, ServiceId := 1);
		nPhase := 3;

	3:
		Ctrl.PackMLIn.eCommand := E_PackMLCommand.Reset;
		Ctrl.PackMLIn.bCommandChangeRequest := TRUE;
		TimelineService(Ctrl := Ctrl, Context := Context, ServiceId := 1);
		nPhase := 4;

	4:
		Ctrl.PackMLIn.bCommandChangeRequest := FALSE;
		TimelineService(Ctrl := Ctrl, Context := Context, ServiceId := 1);
		nPhase := 5;

	5:
		// Keep Starting active for one scan. Its first scan clears all prior history.
		Context.UtcDateTime := '20260916090000000';
		Ctrl.PackMLIn.eCommand := E_PackMLCommand.Start;
		Ctrl.PackMLIn.bCommandChangeRequest := TRUE;
		TimelineService(Ctrl := Ctrl, Context := Context, ServiceId := 1,
			TestExecuteSubState := 1, TestExecuteSubStateName := 'A', StartingBusyScans := 1);
		AssertTrue(Condition := TimelineService.Status.PackMLOut.eStateCurrent =
				E_PackMLState.Starting,
			Message := 'Configured Starting must remain active for one scan.');
		AssertTrue(Condition := (TimelineService.Status.ExecuteSubState.CurrentStep = 0)
				AND (TimelineService.Status.ExecuteSubState.RecordCount = 0)
				AND NOT TimelineService.Status.ExecuteSubState.Overflow,
			Message := 'Entering Starting must clear the Execute substate timeline.');
		nPhase := 6;

	6:
		Context.UtcDateTime := '20260916090100000';
		TimelineService(Ctrl := Ctrl, Context := Context, ServiceId := 1);
		AssertTrue(Condition := (TimelineService.Status.PackMLOut.eStateCurrent =
					E_PackMLState.Execute)
				AND (TimelineService.Status.ExecuteSubState.CurrentStep = 0)
				AND (TimelineService.Status.ExecuteSubState.RecordCount = 0),
			Message :=
				'Starting-to-Execute transition must wait for an evaluated Execute action.');
		nPhase := 7;

	7:
		// The first scan that actually evaluates Execute publishes the first occurrence.
		Context.UtcDateTime := '20260916090200000';
		Ctrl.PackMLIn.bCommandChangeRequest := FALSE;
		TimelineService(Ctrl := Ctrl, Context := Context, ServiceId := 1);
		AssertTrue(Condition := (TimelineService.Status.ExecuteSubState.CurrentStep = 1)
				AND (TimelineService.Status.ExecuteSubState.RecordCount = 1)
				AND (TimelineService.Status.ExecuteSubState.Records[1].Step = 1)
				AND (TimelineService.Status.ExecuteSubState.Records[1].Name = 'A')
				AND (TimelineService.Status.ExecuteSubState.Records[1].StartTimestamp =
					Context.UtcDateTime)
				AND (TimelineService.Status.ExecuteSubState.Records[1].EndTimestamp = ''),
			Message := 'The first evaluated Execute action must open the first occurrence.');
		nPhase := 8;

	8:
		Context.UtcDateTime := '20260916090300000';
		TimelineService(Ctrl := Ctrl, Context := Context, ServiceId := 1,
			TestExecuteSubState := 2, TestExecuteSubStateName := 'B');
		AssertTrue(Condition := (TimelineService.Status.ExecuteSubState.RecordCount = 2)
				AND (TimelineService.Status.ExecuteSubState.Records[1].EndTimestamp =
					Context.UtcDateTime)
				AND (TimelineService.Status.ExecuteSubState.Records[2].StartTimestamp =
					Context.UtcDateTime),
			Message :=
				'A transition must close the old occurrence and open the new one at one timestamp.');
		nPhase := 9;

	9:
		Context.UtcDateTime := '20260916090400000';
		TimelineService(Ctrl := Ctrl, Context := Context, ServiceId := 1,
			TestExecuteSubState := 1, TestExecuteSubStateName := 'A');
		AssertTrue(Condition := (TimelineService.Status.ExecuteSubState.RecordCount = 3)
				AND (TimelineService.Status.ExecuteSubState.Records[3].Step = 1),
			Message := 'Re-entering the same state must append a distinct occurrence.');
		nPhase := 10;

	10:
		Context.UtcDateTime := '20260916090500000';
		Ctrl.PackMLIn.eCommand := E_PackMLCommand.Hold;
		Ctrl.PackMLIn.bCommandChangeRequest := TRUE;
		TimelineService(Ctrl := Ctrl, Context := Context, ServiceId := 1);
		AssertTrue(Condition := (TimelineService.Status.PackMLOut.eStateCurrent =
					E_PackMLState.Held)
				AND (TimelineService.Status.ExecuteSubState.CurrentStep = 0)
				AND (TimelineService.Status.ExecuteSubState.Records[3].EndTimestamp =
					Context.UtcDateTime),
			Message := 'Hold must close the active occurrence while preserving history.');
		nPhase := 11;

	11:
		Ctrl.PackMLIn.bCommandChangeRequest := FALSE;
		TimelineService(Ctrl := Ctrl, Context := Context, ServiceId := 1);
		nPhase := 12;

	12:
		Context.UtcDateTime := '20260916090600000';
		Ctrl.PackMLIn.eCommand := E_PackMLCommand.Unhold;
		Ctrl.PackMLIn.bCommandChangeRequest := TRUE;
		TimelineService(Ctrl := Ctrl, Context := Context, ServiceId := 1);
		AssertTrue(Condition := (TimelineService.Status.PackMLOut.eStateCurrent =
					E_PackMLState.Execute)
				AND (TimelineService.Status.ExecuteSubState.CurrentStep = 0)
				AND (TimelineService.Status.ExecuteSubState.RecordCount = 3),
			Message := 'Unhold transition must wait for an evaluated Execute action.');
		nPhase := 13;

	13:
		Context.UtcDateTime := '20260916090600001';
		Ctrl.PackMLIn.bCommandChangeRequest := FALSE;
		TimelineService(Ctrl := Ctrl, Context := Context, ServiceId := 1);
		AssertTrue(Condition := (TimelineService.Status.ExecuteSubState.CurrentStep = 1)
				AND (TimelineService.Status.ExecuteSubState.RecordCount = 4)
				AND (TimelineService.Status.ExecuteSubState.Records[4].Step = 1)
				AND (TimelineService.Status.ExecuteSubState.Records[4].StartTimestamp =
					Context.UtcDateTime),
			Message :=
				'The first Execute action after Unhold must append the resumed occurrence.');
		nPhase := 14;

	14:
		Context.UtcDateTime := '20260916090700000';
		Ctrl.PackMLIn.eCommand := E_PackMLCommand.Suspend;
		Ctrl.PackMLIn.bCommandChangeRequest := TRUE;
		TimelineService(Ctrl := Ctrl, Context := Context, ServiceId := 1);
		AssertTrue(Condition := (TimelineService.Status.PackMLOut.eStateCurrent =
					E_PackMLState.Suspended)
				AND (TimelineService.Status.ExecuteSubState.CurrentStep = 0)
				AND (TimelineService.Status.ExecuteSubState.Records[4].EndTimestamp =
					Context.UtcDateTime),
			Message := 'Suspend must close the active occurrence.');
		nPhase := 15;

	15:
		Ctrl.PackMLIn.bCommandChangeRequest := FALSE;
		TimelineService(Ctrl := Ctrl, Context := Context, ServiceId := 1);
		nPhase := 16;

	16:
		Context.UtcDateTime := '20260916090800000';
		Ctrl.PackMLIn.eCommand := E_PackMLCommand.Unsuspend;
		Ctrl.PackMLIn.bCommandChangeRequest := TRUE;
		TimelineService(Ctrl := Ctrl, Context := Context, ServiceId := 1);
		AssertTrue(Condition := (TimelineService.Status.PackMLOut.eStateCurrent =
					E_PackMLState.Execute)
				AND (TimelineService.Status.ExecuteSubState.CurrentStep = 0)
				AND (TimelineService.Status.ExecuteSubState.RecordCount = 4),
			Message := 'Unsuspend transition must wait for an evaluated Execute action.');
		nPhase := 17;

	17:
		Context.UtcDateTime := '20260916090800001';
		Ctrl.PackMLIn.bCommandChangeRequest := FALSE;
		TimelineService(Ctrl := Ctrl, Context := Context, ServiceId := 1);
		AssertTrue(Condition := (TimelineService.Status.ExecuteSubState.CurrentStep = 1)
				AND (TimelineService.Status.ExecuteSubState.RecordCount = 5)
				AND (TimelineService.Status.ExecuteSubState.Records[5].Step = 1)
				AND (TimelineService.Status.ExecuteSubState.Records[5].StartTimestamp =
					Context.UtcDateTime),
			Message :=
				'The first Execute action after Unsuspend must append without clearing history.');
		nPhase := 18;

	18:
		Context.UtcDateTime := '20260916090900000';
		TimelineService(
			Ctrl := Ctrl,
			Context := Context,
			ServiceId := 1,
			CompleteExecute := TRUE
		);
		AssertTrue(Condition := (TimelineService.Status.PackMLOut.eStateCurrent =
					E_PackMLState.Completing)
				AND (TimelineService.Status.ExecuteSubState.CurrentStep = 0)
				AND (TimelineService.Status.ExecuteSubState.Records[5].EndTimestamp =
					Context.UtcDateTime),
			Message := 'Natural completion must close the active occurrence.');
		nPhase := 19;

	19:
		TimelineService(
			Ctrl := Ctrl,
			Context := Context,
			ServiceId := 1,
			CompleteExecute := FALSE
		);
		nPhase := 20;

	20:
		Ctrl.PackMLIn.eCommand := E_PackMLCommand.Reset;
		Ctrl.PackMLIn.bCommandChangeRequest := TRUE;
		TimelineService(Ctrl := Ctrl, Context := Context, ServiceId := 1);
		nPhase := 21;

	21:
		Ctrl.PackMLIn.bCommandChangeRequest := FALSE;
		TimelineService(Ctrl := Ctrl, Context := Context, ServiceId := 1);
		nPhase := 22;

	22:
		// This Starting completes in the same scan. It clears history but does not sample Execute yet.
		Context.UtcDateTime := '20260916091000000';
		Ctrl.PackMLIn.eCommand := E_PackMLCommand.Start;
		Ctrl.PackMLIn.bCommandChangeRequest := TRUE;
		TimelineService(Ctrl := Ctrl, Context := Context, ServiceId := 1,
			TestExecuteSubState := 2, TestExecuteSubStateName := 'B', StartingBusyScans := 0);
		AssertTrue(Condition := (TimelineService.Status.PackMLOut.eStateCurrent =
					E_PackMLState.Execute)
				AND (TimelineService.Status.ExecuteSubState.CurrentStep = 0)
				AND (TimelineService.Status.ExecuteSubState.RecordCount = 0)
				AND NOT TimelineService.Status.ExecuteSubState.Overflow
				AND (TimelineService.Status.ExecuteSubState.Records[1].Step = 0),
			Message := 'Same-scan Starting must clear history and defer Execute sampling.');
		nPhase := 23;

	23:
		Context.UtcDateTime := '20260916091000001';
		Ctrl.PackMLIn.bCommandChangeRequest := FALSE;
		TimelineService(Ctrl := Ctrl, Context := Context, ServiceId := 1);
		AssertTrue(Condition := (TimelineService.Status.ExecuteSubState.CurrentStep = 2)
				AND (TimelineService.Status.ExecuteSubState.RecordCount = 1)
				AND (TimelineService.Status.ExecuteSubState.Records[1].Step = 2)
				AND (TimelineService.Status.ExecuteSubState.Records[1].StartTimestamp =
					Context.UtcDateTime)
				AND (TimelineService.Status.ExecuteSubState.Records[2].Step = 0),
			Message := 'The next Execute action must record the first substate of the new run.');
		nPhase := 24;

	24:
		Context.UtcDateTime := '20260916091100000';
		Ctrl.PackMLIn.eCommand := E_PackMLCommand.Stop;
		Ctrl.PackMLIn.bCommandChangeRequest := TRUE;
		TimelineService(Ctrl := Ctrl, Context := Context, ServiceId := 1);
		AssertTrue(Condition := (TimelineService.Status.PackMLOut.eStateCurrent =
					E_PackMLState.Stopped)
				AND (TimelineService.Status.ExecuteSubState.CurrentStep = 0)
				AND (TimelineService.Status.ExecuteSubState.Records[1].EndTimestamp =
					Context.UtcDateTime),
			Message := 'Stop must close the active occurrence.');
		nPhase := 25;

	25:
		Ctrl.PackMLIn.bCommandChangeRequest := FALSE;
		TimelineService(Ctrl := Ctrl, Context := Context, ServiceId := 1);
		nPhase := 26;

	26:
		Ctrl.PackMLIn.eCommand := E_PackMLCommand.Reset;
		Ctrl.PackMLIn.bCommandChangeRequest := TRUE;
		TimelineService(Ctrl := Ctrl, Context := Context, ServiceId := 1);
		nPhase := 27;

	27:
		Ctrl.PackMLIn.bCommandChangeRequest := FALSE;
		TimelineService(Ctrl := Ctrl, Context := Context, ServiceId := 1);
		nPhase := 28;

	28:
		Context.UtcDateTime := '20260916091200000';
		Ctrl.PackMLIn.eCommand := E_PackMLCommand.Start;
		Ctrl.PackMLIn.bCommandChangeRequest := TRUE;
		TimelineService(Ctrl := Ctrl, Context := Context, ServiceId := 1,
			TestExecuteSubState := 3, TestExecuteSubStateName := 'C');
		nPhase := 29;

	29:
		Ctrl.PackMLIn.bCommandChangeRequest := FALSE;
		TimelineService(Ctrl := Ctrl, Context := Context, ServiceId := 1);
		nPhase := 30;

	30:
		Context.UtcDateTime := '20260916091300000';
		Ctrl.PackMLIn.eCommand := E_PackMLCommand.Abort;
		Ctrl.PackMLIn.bCommandChangeRequest := TRUE;
		TimelineService(Ctrl := Ctrl, Context := Context, ServiceId := 1);
		AssertTrue(Condition := (TimelineService.Status.PackMLOut.eStateCurrent =
					E_PackMLState.Aborted)
				AND (TimelineService.Status.ExecuteSubState.CurrentStep = 0)
				AND (TimelineService.Status.ExecuteSubState.Records[1].EndTimestamp =
					Context.UtcDateTime),
			Message := 'Abort must close the active occurrence.');
		nPhase := 0;
		TEST_FINISHED();
END_CASE
END_METHOD

END_FUNCTION_BLOCK

// ---- Fakes/FB_TestableCarryoverSubStateService.TcPOU
FUNCTION_BLOCK FB_TestableCarryoverSubStateService EXTENDS FB_ServiceBase
VAR
	// Simulate a second run that still holds the previous run's final substate.
	_Step : UDINT := 5;
END_VAR

M_UpdateService(CompletionBehavior := E_ServiceCompletionBehavior.NaturalCompletion);

METHOD PROTECTED H_GetExecuteSubState : UDINT
H_GetExecuteSubState := _Step;
END_METHOD

METHOD PROTECTED H_GetExecuteSubStateName : STRING(80)
CASE _Step OF
	1: H_GetExecuteSubStateName := 'LiftReady';
	5: H_GetExecuteSubStateName := 'Finish';
ELSE
	H_GetExecuteSubStateName := '';
END_CASE
END_METHOD

METHOD PROTECTED H_OnExecute : E_PackMLHookResult
VAR_INPUT
	bFirstScan : BOOL;
END_VAR
IF bFirstScan THEN
	_Step := 1;
END_IF
H_OnExecute := E_PackMLHookResult.Busy;
END_METHOD

END_FUNCTION_BLOCK

// ---- POUs/Test Suites/Service/FB_CompositeServiceBaseTests.TcPOU
FUNCTION_BLOCK FB_CompositeServiceBaseTests EXTENDS TcUnit.FB_TestSuite

DefinitionRegistersOnceAndOnlyInsideDeclarationWindow();
UnconfiguredCompositeStartStopsWithFrameworkError();

METHOD DefinitionRegistersOnceAndOnlyInsideDeclarationWindow
VAR_INST
	Composite : FB_TestCompositeService;
	Coordinator : FB_ServiceCoordinator;
	CompositeUpperCtrl : ST_ServiceCtrl;
	CompositeEffectiveCtrl : ST_ServiceCtrl;
	CompositeUpperParam : ST_TestServiceParam;
	CompositeEffectiveParam : ST_TestServiceParam;
	CompositeStatus : ST_ServiceStatus;
	ChildUpperCtrl : ST_ServiceCtrl;
	ChildEffectiveCtrl : ST_ServiceCtrl;
	ChildUpperParam : ST_TestServiceParam;
	ChildEffectiveParam : ST_TestServiceParam;
	ChildStatus : ST_ServiceStatus;
END_VAR
TEST('DefinitionRegistersOnceAndOnlyInsideDeclarationWindow');

// Arrange：先登錄 Composite 本身與允許 Composite 呼叫的 dependency。
Coordinator.M_BeginRegistration();
AssertTrue(
	Condition := Coordinator.M_Register(
		ServiceId := 10,
		AllowCompositeCall := FALSE,
		UpperCtrl := CompositeUpperCtrl,
		EffectiveCtrl := CompositeEffectiveCtrl,
		UpperParam := CompositeUpperParam,
		EffectiveParam := CompositeEffectiveParam,
		Status := CompositeStatus
	),
	Message := 'Composite Service storage must register.'
);
AssertTrue(
	Condition := Coordinator.M_Register(
		ServiceId := 20,
		AllowCompositeCall := TRUE,
		UpperCtrl := ChildUpperCtrl,
		EffectiveCtrl := ChildEffectiveCtrl,
		UpperParam := ChildUpperParam,
		EffectiveParam := ChildEffectiveParam,
		Status := ChildStatus
	),
	Message := 'Dependency Service storage must register.'
);
Composite.DependencyCount := 1;
Composite.DependencyOne := 20;

// Act / Assert：definition 僅可成功一次，且 M_AddDependency 不能在 hook 之外使用。
AssertTrue(
	Condition := Composite.M_RegisterDefinition(
		CompositeServiceId := 10,
		Coordinator := Coordinator
	),
	Message := 'First valid Composite definition must register.'
);
AssertFalse(
	Condition := Composite.M_RegisterDefinition(
		CompositeServiceId := 10,
		Coordinator := Coordinator
	),
	Message := 'Composite definition must be one-shot.'
);
AssertFalse(
	Condition := Composite.M_TestAddDependencyOutsideDefinition(ServiceIdValue := 20),
	Message := 'Dependency declaration must be restricted to H_DeclareServices.'
);

TEST_FINISHED();
END_METHOD

METHOD UnconfiguredCompositeStartStopsWithFrameworkError
VAR_INST
	Composite : FB_TestCompositeService;
	Ctrl : ST_ServiceCtrl;
	Context : ST_ServiceContext;
	nPhase : UINT;
END_VAR
TEST('UnconfiguredCompositeStartStopsWithFrameworkError');

